screen "78_3BR" 800x454, template "Template_1"
   on GenerateScreen: SetTag("Tag_ScreenNumber", 78)
   TextField "Text field_1" at 17,28 size 250x21; Text 'Слово керування енкодером:'
   Circle "Circle_1" at 28,55 size 16x16
      Appearance <- "STW2_ENC"
   Circle "Circle_2" at 28,75 size 16x16
      Appearance <- "ZSW2_ENC"
   Circle "Circle_3" at 28,95 size 16x16
      Appearance <- "STW2_ENC"
   TextField "Text field_3" at 56,54 size 231x18; Text 'Трігер на калібровку енкодера'
   TextField "Text field_4" at 56,74 size 154x18; Text 'Квитування помилки'
   TextField "Text field_5" at 56,94 size 123x18; Text 'Контроль з PLC'
   IOField "I/O field_1" at 16,115 size 40x20; FormatPattern FFFF
      ProcessValue <- "STW2_ENC"
   TextField "Text field_6" at 56,115 size 248x18; Text 'Сигнал працездатності енкодера'
   TextField "Text field_12" at 403,28 size 210x21; Text 'Слово статусу енкодера:'
   Circle "Circle_9" at 414,55 size 16x16
      Appearance <- "ZSW2_ENC"
   TextField "Text field_14" at 442,54 size 350x18; Text 'Підтвердження встановлення нового значення'
   Circle "Circle_10" at 414,75 size 16x16
      Appearance <- "ZSW2_ENC"
   TextField "Text field_15" at 442,74 size 234x18; Text 'Фактичне положення є дійсним'
   Circle "Circle_11" at 414,95 size 16x16
      Appearance <- "ZSW2_ENC"
   TextField "Text field_16" at 442,94 size 228x18; Text 'Фактична швидкість є дійсною'
   Circle "Circle_12" at 414,115 size 16x16
      Appearance <- "ZSW2_ENC"
   TextField "Text field_17" at 442,114 size 129x18; Text 'Помилка активна'
   Circle "Circle_13" at 414,135 size 16x16
      Appearance <- "ZSW2_ENC"
   TextField "Text field_18" at 442,134 size 176x18; Text 'Попередження активне'
   Circle "Circle_14" at 414,155 size 16x16
      Appearance <- "ZSW2_ENC"
   TextField "Text field_19" at 442,154 size 145x18; Text 'Запит на перевірку'
   TextField "Text field_20" at 442,174 size 248x18; Text 'Сигнал працездатності енкодера'
   IOField "I/O field_2" at 402,173 size 40x20; FormatPattern FFFF
      ProcessValue <- "ZSW2_ENC"
   IOField "I/O field_3" at 148,364 size 70x20; FormatPattern s9999999999
      ProcessValue <- "RawPosition"
   TextField "Text field_26" at 28,363 size 107x21; Text 'Положення:'
   IOField "I/O field_4" at 534,364 size 70x20; FormatPattern s9999999999
      ProcessValue <- "RawVelocity"
   TextField "Text field_27" at 414,363 size 97x21; Text 'Швидкість:'
   Circle "Circle_4" at 28,222 size 16x16
      Appearance <- "EncoderLifeValid"
   TextField "Text field_2" at 56,221 size 228x18; Text 'Sign-of-life енкодера валідний'
   Circle "Circle_5" at 28,242 size 16x16
      Appearance <- "EncoderReady"
   TextField "Text field_7" at 56,241 size 325x18; Text 'Енкодер готовий для використання в логіці'
   Circle "Circle_6" at 28,262 size 16x16
      Appearance <- "CommunicationFault"
   TextField "Text field_8" at 56,261 size 288x18; Text 'Загальна помилка обміну з енкодером'
   Circle "Circle_7" at 28,282 size 16x16
      Appearance <- "PresetBusy"
   TextField "Text field_9" at 56,281 size 198x18; Text 'Preset-процедура активна'
   Circle "Circle_8" at 28,302 size 16x16
      Appearance <- "PresetDone"
   TextField "Text field_10" at 56,301 size 191x18; Text 'Preset успішно виконано.'
   Circle "Circle_15" at 28,322 size 16x16
      Appearance <- "PresetError"
   TextField "Text field_11" at 56,321 size 198x18; Text 'Помилка виконання preset'
   TextField "Text field_13" at 414,249 size 127x18; Text 'Статус енкодеру'
   TextField "Text field_21" at 414,221 size 115x18; Text 'Статус пресету'
   SymbolicIOField "Symbolic I/O field_1" at 562,214 size 230x32; TextOff '0'; TextOn '1'; TextList "PresetStatus"
      ProcessValue <- "PresetStatus"
   SymbolicIOField "Symbolic I/O field_2" at 562,242 size 230x32; TextOff '0'; TextOn '1'; TextList "EncoderStatus"
      ProcessValue <- "Status"
   TextField "Text field_22" at 308,6 size 185x23; Text 'Стан енкодеру 3BR'

screen "79_4BR1" 800x454, template "Template_1"
   on GenerateScreen: SetTag("Tag_ScreenNumber", 79)
   TextField "Text field_1" at 17,28 size 250x21; Text 'Слово керування енкодером:'
   Circle "Circle_1" at 28,55 size 16x16
      Appearance <- "STW2_ENC"
   Circle "Circle_2" at 28,75 size 16x16
      Appearance <- "ZSW2_ENC"
   Circle "Circle_3" at 28,95 size 16x16
      Appearance <- "STW2_ENC"
   TextField "Text field_3" at 56,54 size 231x18; Text 'Трігер на калібровку енкодера'
   TextField "Text field_4" at 56,74 size 154x18; Text 'Квитування помилки'
   TextField "Text field_5" at 56,94 size 123x18; Text 'Контроль з PLC'
   IOField "I/O field_1" at 16,115 size 40x20; FormatPattern FFFF
      ProcessValue <- "STW2_ENC"
   TextField "Text field_6" at 56,115 size 248x18; Text 'Сигнал працездатності енкодера'
   TextField "Text field_12" at 403,28 size 210x21; Text 'Слово статусу енкодера:'
   Circle "Circle_9" at 414,55 size 16x16
      Appearance <- "ZSW2_ENC"
   TextField "Text field_14" at 442,54 size 350x18; Text 'Підтвердження встановлення нового значення'
   Circle "Circle_10" at 414,75 size 16x16
      Appearance <- "ZSW2_ENC"
   TextField "Text field_15" at 442,74 size 234x18; Text 'Фактичне положення є дійсним'
   Circle "Circle_11" at 414,95 size 16x16
      Appearance <- "ZSW2_ENC"
   TextField "Text field_16" at 442,94 size 228x18; Text 'Фактична швидкість є дійсною'
   Circle "Circle_12" at 414,115 size 16x16
      Appearance <- "ZSW2_ENC"
   TextField "Text field_17" at 442,114 size 129x18; Text 'Помилка активна'
   Circle "Circle_13" at 414,135 size 16x16
      Appearance <- "ZSW2_ENC"
   TextField "Text field_18" at 442,134 size 176x18; Text 'Попередження активне'
   Circle "Circle_14" at 414,155 size 16x16
      Appearance <- "ZSW2_ENC"
   TextField "Text field_19" at 442,154 size 145x18; Text 'Запит на перевірку'
   TextField "Text field_20" at 442,174 size 248x18; Text 'Сигнал працездатності енкодера'
   IOField "I/O field_2" at 402,173 size 40x20; FormatPattern FFFF
      ProcessValue <- "ZSW2_ENC"
   IOField "I/O field_3" at 148,364 size 70x20; FormatPattern s9999999999
      ProcessValue <- "RawPosition"
   TextField "Text field_26" at 28,363 size 107x21; Text 'Положення:'
   IOField "I/O field_4" at 534,364 size 70x20; FormatPattern s9999999999
      ProcessValue <- "RawVelocity"
   TextField "Text field_27" at 414,363 size 97x21; Text 'Швидкість:'
   Circle "Circle_4" at 28,222 size 16x16
      Appearance <- "EncoderLifeValid"
   TextField "Text field_2" at 56,221 size 228x18; Text 'Sign-of-life енкодера валідний'
   Circle "Circle_5" at 28,242 size 16x16
      Appearance <- "EncoderReady"
   TextField "Text field_7" at 56,241 size 325x18; Text 'Енкодер готовий для використання в логіці'
   Circle "Circle_6" at 28,262 size 16x16
      Appearance <- "CommunicationFault"
   TextField "Text field_8" at 56,261 size 288x18; Text 'Загальна помилка обміну з енкодером'
   Circle "Circle_7" at 28,282 size 16x16
      Appearance <- "PresetBusy"
   TextField "Text field_9" at 56,281 size 198x18; Text 'Preset-процедура активна'
   Circle "Circle_8" at 28,302 size 16x16
      Appearance <- "PresetDone"
   TextField "Text field_10" at 56,301 size 191x18; Text 'Preset успішно виконано.'
   Circle "Circle_15" at 28,322 size 16x16
      Appearance <- "PresetError"
   TextField "Text field_11" at 56,321 size 198x18; Text 'Помилка виконання preset'
   TextField "Text field_13" at 414,249 size 127x18; Text 'Статус енкодеру'
   TextField "Text field_21" at 414,221 size 115x18; Text 'Статус пресету'
   SymbolicIOField "Symbolic I/O field_1" at 562,214 size 230x32; TextOff '0'; TextOn '1'; TextList "PresetStatus"
      ProcessValue <- "PresetStatus"
   SymbolicIOField "Symbolic I/O field_2" at 562,242 size 230x32; TextOff '0'; TextOn '1'; TextList "EncoderStatus"
      ProcessValue <- "Status"
   TextField "Text field_22" at 308,6 size 196x23; Text 'Стан енкодеру 4BR1'

screen "710_4BR2" 800x454, template "Template_1"
   on GenerateScreen: SetTag("Tag_ScreenNumber", 710)
   TextField "Text field_1" at 17,28 size 250x21; Text 'Слово керування енкодером:'
   Circle "Circle_1" at 28,55 size 16x16
      Appearance <- "STW2_ENC"
   Circle "Circle_2" at 28,75 size 16x16
      Appearance <- "ZSW2_ENC"
   Circle "Circle_3" at 28,95 size 16x16
      Appearance <- "STW2_ENC"
   TextField "Text field_3" at 56,54 size 231x18; Text 'Трігер на калібровку енкодера'
   TextField "Text field_4" at 56,74 size 154x18; Text 'Квитування помилки'
   TextField "Text field_5" at 56,94 size 123x18; Text 'Контроль з PLC'
   IOField "I/O field_1" at 16,115 size 40x20; FormatPattern FFFF
      ProcessValue <- "STW2_ENC"
   TextField "Text field_6" at 56,115 size 248x18; Text 'Сигнал працездатності енкодера'
   TextField "Text field_12" at 403,28 size 210x21; Text 'Слово статусу енкодера:'
   Circle "Circle_9" at 414,55 size 16x16
      Appearance <- "ZSW2_ENC"
   TextField "Text field_14" at 442,54 size 350x18; Text 'Підтвердження встановлення нового значення'
   Circle "Circle_10" at 414,75 size 16x16
      Appearance <- "ZSW2_ENC"
   TextField "Text field_15" at 442,74 size 234x18; Text 'Фактичне положення є дійсним'
   Circle "Circle_11" at 414,95 size 16x16
      Appearance <- "ZSW2_ENC"
   TextField "Text field_16" at 442,94 size 228x18; Text 'Фактична швидкість є дійсною'
   Circle "Circle_12" at 414,115 size 16x16
      Appearance <- "ZSW2_ENC"
   TextField "Text field_17" at 442,114 size 129x18; Text 'Помилка активна'
   Circle "Circle_13" at 414,135 size 16x16
      Appearance <- "ZSW2_ENC"
   TextField "Text field_18" at 442,134 size 176x18; Text 'Попередження активне'
   Circle "Circle_14" at 414,155 size 16x16
      Appearance <- "ZSW2_ENC"
   TextField "Text field_19" at 442,154 size 145x18; Text 'Запит на перевірку'
   TextField "Text field_20" at 442,174 size 248x18; Text 'Сигнал працездатності енкодера'
   IOField "I/O field_2" at 402,173 size 40x20; FormatPattern FFFF
      ProcessValue <- "ZSW2_ENC"
   IOField "I/O field_3" at 148,364 size 70x20; FormatPattern s9999999999
      ProcessValue <- "RawPosition"
   TextField "Text field_26" at 28,363 size 107x21; Text 'Положення:'
   IOField "I/O field_4" at 534,364 size 70x20; FormatPattern s9999999999
      ProcessValue <- "RawVelocity"
   TextField "Text field_27" at 414,363 size 97x21; Text 'Швидкість:'
   Circle "Circle_4" at 28,222 size 16x16
      Appearance <- "EncoderLifeValid"
   TextField "Text field_2" at 56,221 size 228x18; Text 'Sign-of-life енкодера валідний'
   Circle "Circle_5" at 28,242 size 16x16
      Appearance <- "EncoderReady"
   TextField "Text field_7" at 56,241 size 325x18; Text 'Енкодер готовий для використання в логіці'
   Circle "Circle_6" at 28,262 size 16x16
      Appearance <- "CommunicationFault"
   TextField "Text field_8" at 56,261 size 288x18; Text 'Загальна помилка обміну з енкодером'
   Circle "Circle_7" at 28,282 size 16x16
      Appearance <- "PresetBusy"
   TextField "Text field_9" at 56,281 size 198x18; Text 'Preset-процедура активна'
   Circle "Circle_8" at 28,302 size 16x16
      Appearance <- "PresetDone"
   TextField "Text field_10" at 56,301 size 191x18; Text 'Preset успішно виконано.'
   Circle "Circle_15" at 28,322 size 16x16
      Appearance <- "PresetError"
   TextField "Text field_11" at 56,321 size 198x18; Text 'Помилка виконання preset'
   TextField "Text field_13" at 414,249 size 127x18; Text 'Статус енкодеру'
   TextField "Text field_21" at 414,221 size 115x18; Text 'Статус пресету'
   SymbolicIOField "Symbolic I/O field_1" at 562,214 size 230x32; TextOff '0'; TextOn '1'; TextList "PresetStatus"
      ProcessValue <- "PresetStatus"
   SymbolicIOField "Symbolic I/O field_2" at 562,242 size 230x32; TextOff '0'; TextOn '1'; TextList "EncoderStatus"
      ProcessValue <- "Status"
   TextField "Text field_22" at 308,6 size 196x23; Text 'Стан енкодеру 4BR2'

screen "61_Архіви(3UZ1)" 800x454, template "Template_1"
   on GenerateScreen: SetTag("Tag_ScreenNumber", 61); SetTag("iVisibilityDevices", 0)
   Button "btnLiftUp" at 8,120 size 96x32; TextOff '3UZ1'
   Button "btnTrolley" at 8,160 size 96x32; TextOff '4UZ1'
      on Release: ActivateScreen("62_Архіви(4UZ1)", 0)
   Button "btnCrane" at 8,200 size 96x32; TextOff '4UZ2'
      on Release: ActivateScreen("63_Архіви(4UZ2)", 0)
   Button "btnContactor" at 8,80 size 96x32; TextOff '1UZ1'
      on Release: ActivateScreen("60_Архіви(1UZ1)", 0)
   Button "Button_1" at 8,319 size 96x32; TextOff 'Струм Момент'
      on Release: SetTag("iVisibilityDevices", 0)
      Appearance <- "iVisibilityDevices"
   Button "Button_2" at 8,356 size 96x32; TextOff 'Швидкості'
      on Release: SetTag("iVisibilityDevices", 1)
      Appearance <- "iVisibilityDevices"
   TrendView "trvCurrent" at 155,10 size 640x200
      Visibility <- "iVisibilityDevices"
   TrendView "trvMoment" at 155,208 size 640x200
      Visibility <- "iVisibilityDevices"
   TextField "txtCurrent" at 125,95 size 19x30; Text 'I ,А'
      Visibility <- "iVisibilityDevices"
   TextField "txtMoment" at 125,278 size 19x60; Text 'M , Н*м'
      Visibility <- "iVisibilityDevices"
   Button "btnCurrentDoubleBack" at 111,10 size 40x20; TextOff 'Text'; PictureOff "FB_2ArrowsLeft_Rectangular_Released_256c"; PictureOn "FB_2ArrowsLeft_Rectangular_Pressed_256c"
      on Press: function_f26ff0ec("trvCurrent")
      on Release: function_f26ff0ec("trvCurrent")
      Visibility <- "iVisibilityDevices"
   Button "btnCurrentOneBack" at 111,35 size 40x20; TextOff 'Text'; PictureOff "FB_ArrowLeft_Rectangular_Released_256c"; PictureOn "FB_ArrowLeft_Rectangular_Pressed_256c"
      on Press: function_f26ff0ec("trvCurrent")
      Visibility <- "iVisibilityDevices"
   Button "btnCurrentForward" at 111,149 size 40x20; TextOff 'Text'; PictureOff "FB_ArrowRight_Rectangular_Released_256c"; PictureOn "FB_ArrowRight_Rectangular_Pressed_256c"
      on Press: function_c2ce674d("trvCurrent")
      Visibility <- "iVisibilityDevices"
   Button "btnCurrentDoubleForward" at 111,174 size 40x20; TextOff 'Text'; PictureOff "FB_2ArrowsRight_Rectangular_Released_256c"; PictureOn "FB_2ArrowsRight_Rectangular_Pressed_256c"
      on Press: function_c2ce674d("trvCurrent")
      on Release: function_c2ce674d("trvCurrent")
      Visibility <- "iVisibilityDevices"
   Button "btnMomentDoubleBack" at 111,208 size 40x20; TextOff 'Text'; PictureOff "FB_2ArrowsLeft_Rectangular_Released_256c"; PictureOn "FB_2ArrowsLeft_Rectangular_Pressed_256c"
      on Press: function_f26ff0ec("trvMoment")
      on Release: function_f26ff0ec("trvMoment")
      Visibility <- "iVisibilityDevices"
   Button "btnMomentOneBack" at 111,233 size 40x20; TextOff 'Text'; PictureOff "FB_ArrowLeft_Rectangular_Released_256c"; PictureOn "FB_ArrowLeft_Rectangular_Pressed_256c"
      on Press: function_f26ff0ec("trvMoment")
      Visibility <- "iVisibilityDevices"
   Button "btnMomentOneForward" at 111,363 size 40x20; TextOff 'Text'; PictureOff "FB_ArrowRight_Rectangular_Released_256c"; PictureOn "FB_ArrowRight_Rectangular_Pressed_256c"
      on Press: function_c2ce674d("trvMoment")
      Visibility <- "iVisibilityDevices"
   Button "btnMomentDoubleForward" at 111,388 size 40x20; TextOff 'Text'; PictureOff "FB_2ArrowsRight_Rectangular_Released_256c"; PictureOn "FB_2ArrowsRight_Rectangular_Pressed_256c"
      on Press: function_c2ce674d("trvMoment")
      on Release: function_c2ce674d("trvMoment")
      Visibility <- "iVisibilityDevices"
   TrendView "trvSpeed" at 155,10 size 640x200
      Visibility <- "iVisibilityDevices"
   TrendView "trvError" at 155,208 size 640x200
      Visibility <- "iVisibilityDevices"
   TextField "txtSpeed" at 108,84 size 19x53; Text 'W_set,'
      Visibility <- "iVisibilityDevices"
   TextField "txtError" at 125,259 size 19x98; Text 'W_err ,об/хв'
      Visibility <- "iVisibilityDevices"
   TextField "txtSpeed_1" at 120,82 size 19x57; Text 'W_real,'
      Visibility <- "iVisibilityDevices"
   TextField "txtSpeed_2" at 132,87 size 19x46; Text 'об/хв'
      Visibility <- "iVisibilityDevices"
   Button "btnSpeedDoubleBack" at 111,10 size 40x20; TextOff 'Text'; PictureOff "FB_2ArrowsLeft_Rectangular_Released_256c"; PictureOn "FB_2ArrowsLeft_Rectangular_Pressed_256c"
      on Press: function_f26ff0ec("trvSpeed")
      on Release: function_f26ff0ec("trvSpeed")
      Visibility <- "iVisibilityDevices"
   Button "btnSpeedOneBack" at 111,35 size 40x20; TextOff 'Text'; PictureOff "FB_ArrowLeft_Rectangular_Released_256c"; PictureOn "FB_ArrowLeft_Rectangular_Pressed_256c"
      on Press: function_f26ff0ec("trvSpeed")
      Visibility <- "iVisibilityDevices"
   Button "btnSpeedForward" at 111,149 size 40x20; TextOff 'Text'; PictureOff "FB_ArrowRight_Rectangular_Released_256c"; PictureOn "FB_ArrowRight_Rectangular_Pressed_256c"
      on Press: function_c2ce674d("trvSpeed")
      Visibility <- "iVisibilityDevices"
   Button "btnSpeedDoubleForward" at 111,174 size 40x20; TextOff 'Text'; PictureOff "FB_2ArrowsRight_Rectangular_Released_256c"; PictureOn "FB_2ArrowsRight_Rectangular_Pressed_256c"
      on Press: function_c2ce674d("trvSpeed")
      on Release: function_c2ce674d("trvSpeed")
      Visibility <- "iVisibilityDevices"
   Button "btnErrorDoubleBack" at 111,208 size 40x20; TextOff 'Text'; PictureOff "FB_2ArrowsLeft_Rectangular_Released_256c"; PictureOn "FB_2ArrowsLeft_Rectangular_Pressed_256c"
      on Press: function_f26ff0ec("trvError")
      on Release: function_f26ff0ec("trvError")
      Visibility <- "iVisibilityDevices"
   Button "btnErrorOneBack" at 111,233 size 40x20; TextOff 'Text'; PictureOff "FB_ArrowLeft_Rectangular_Released_256c"; PictureOn "FB_ArrowLeft_Rectangular_Pressed_256c"
      on Press: function_f26ff0ec("trvError")
      Visibility <- "iVisibilityDevices"
   Button "btnErrorOneForward" at 111,363 size 40x20; TextOff 'Text'; PictureOff "FB_ArrowRight_Rectangular_Released_256c"; PictureOn "FB_ArrowRight_Rectangular_Pressed_256c"
      on Press: function_c2ce674d("trvError")
      Visibility <- "iVisibilityDevices"
   Button "btnErrorDoubleForward" at 111,388 size 40x20; TextOff 'Text'; PictureOff "FB_2ArrowsRight_Rectangular_Released_256c"; PictureOn "FB_2ArrowsRight_Rectangular_Pressed_256c"
      on Press: function_c2ce674d("trvError")
      on Release: function_c2ce674d("trvError")
      Visibility <- "iVisibilityDevices"

screen "62_Архіви(4UZ1)" 800x454, template "Template_1"
   on GenerateScreen: SetTag("Tag_ScreenNumber", 62); SetTag("iVisibilityDevices", 0)
   Button "btnLiftUp" at 8,120 size 96x32; TextOff '3UZ1'
      on Release: ActivateScreen("61_Архіви(3UZ1)", 0)
   Button "btnTrolley" at 8,160 size 96x32; TextOff '4UZ1'
   Button "btnCrane" at 8,200 size 96x32; TextOff '4UZ2'
      on Release: ActivateScreen("63_Архіви(4UZ2)", 0)
   Button "btnContactor" at 8,80 size 96x32; TextOff '1UZ1'
      on Release: ActivateScreen("60_Архіви(1UZ1)", 0)
   Button "Button_1" at 8,319 size 96x32; TextOff 'Струм Момент'
      on Release: SetTag("iVisibilityDevices", 0)
      Appearance <- "iVisibilityDevices"
   Button "Button_2" at 8,356 size 96x32; TextOff 'Швидкості'
      on Release: SetTag("iVisibilityDevices", 1)
      Appearance <- "iVisibilityDevices"
   TrendView "trvCurrent" at 155,10 size 640x200
      Visibility <- "iVisibilityDevices"
   TrendView "trvMoment" at 155,208 size 640x200
      Visibility <- "iVisibilityDevices"
   TextField "txtCurrent" at 125,95 size 19x30; Text 'I ,А'
      Visibility <- "iVisibilityDevices"
   TextField "txtMoment" at 125,278 size 19x60; Text 'M , Н*м'
      Visibility <- "iVisibilityDevices"
   Button "btnCurrentDoubleBack" at 111,10 size 40x20; TextOff 'Text'; PictureOff "FB_2ArrowsLeft_Rectangular_Released_256c"; PictureOn "FB_2ArrowsLeft_Rectangular_Pressed_256c"
      on Press: function_f26ff0ec("trvCurrent")
      on Release: function_f26ff0ec("trvCurrent")
      Visibility <- "iVisibilityDevices"
   Button "btnCurrentOneBack" at 111,35 size 40x20; TextOff 'Text'; PictureOff "FB_ArrowLeft_Rectangular_Released_256c"; PictureOn "FB_ArrowLeft_Rectangular_Pressed_256c"
      on Press: function_f26ff0ec("trvCurrent")
      Visibility <- "iVisibilityDevices"
   Button "btnCurrentForward" at 111,149 size 40x20; TextOff 'Text'; PictureOff "FB_ArrowRight_Rectangular_Released_256c"; PictureOn "FB_ArrowRight_Rectangular_Pressed_256c"
      on Press: function_c2ce674d("trvCurrent")
      Visibility <- "iVisibilityDevices"
   Button "btnCurrentDoubleForward" at 111,174 size 40x20; TextOff 'Text'; PictureOff "FB_2ArrowsRight_Rectangular_Released_256c"; PictureOn "FB_2ArrowsRight_Rectangular_Pressed_256c"
      on Press: function_c2ce674d("trvCurrent")
      on Release: function_c2ce674d("trvCurrent")
      Visibility <- "iVisibilityDevices"
   Button "btnMomentDoubleBack" at 111,208 size 40x20; TextOff 'Text'; PictureOff "FB_2ArrowsLeft_Rectangular_Released_256c"; PictureOn "FB_2ArrowsLeft_Rectangular_Pressed_256c"
      on Press: function_f26ff0ec("trvMoment")
      on Release: function_f26ff0ec("trvMoment")
      Visibility <- "iVisibilityDevices"
   Button "btnMomentOneBack" at 111,233 size 40x20; TextOff 'Text'; PictureOff "FB_ArrowLeft_Rectangular_Released_256c"; PictureOn "FB_ArrowLeft_Rectangular_Pressed_256c"
      on Press: function_f26ff0ec("trvMoment")
      Visibility <- "iVisibilityDevices"
   Button "btnMomentOneForward" at 111,363 size 40x20; TextOff 'Text'; PictureOff "FB_ArrowRight_Rectangular_Released_256c"; PictureOn "FB_ArrowRight_Rectangular_Pressed_256c"
      on Press: function_c2ce674d("trvMoment")
      Visibility <- "iVisibilityDevices"
   Button "btnMomentDoubleForward" at 111,388 size 40x20; TextOff 'Text'; PictureOff "FB_2ArrowsRight_Rectangular_Released_256c"; PictureOn "FB_2ArrowsRight_Rectangular_Pressed_256c"
      on Press: function_c2ce674d("trvMoment")
      on Release: function_c2ce674d("trvMoment")
      Visibility <- "iVisibilityDevices"
   TrendView "trvSpeed" at 155,10 size 640x200
      Visibility <- "iVisibilityDevices"
   TrendView "trvError" at 155,208 size 640x200
      Visibility <- "iVisibilityDevices"
   TextField "txtSpeed" at 108,84 size 19x53; Text 'W_set,'
      Visibility <- "iVisibilityDevices"
   TextField "txtError" at 125,259 size 19x98; Text 'W_err ,об/хв'
      Visibility <- "iVisibilityDevices"
   TextField "txtSpeed_1" at 120,82 size 19x57; Text 'W_real,'
      Visibility <- "iVisibilityDevices"
   TextField "txtSpeed_2" at 132,87 size 19x46; Text 'об/хв'
      Visibility <- "iVisibilityDevices"
   Button "btnSpeedDoubleBack" at 111,10 size 40x20; TextOff 'Text'; PictureOff "FB_2ArrowsLeft_Rectangular_Released_256c"; PictureOn "FB_2ArrowsLeft_Rectangular_Pressed_256c"
      on Press: function_f26ff0ec("trvSpeed")
      on Release: function_f26ff0ec("trvSpeed")
      Visibility <- "iVisibilityDevices"
   Button "btnSpeedOneBack" at 111,35 size 40x20; TextOff 'Text'; PictureOff "FB_ArrowLeft_Rectangular_Released_256c"; PictureOn "FB_ArrowLeft_Rectangular_Pressed_256c"
      on Press: function_f26ff0ec("trvSpeed")
      Visibility <- "iVisibilityDevices"
   Button "btnSpeedForward" at 111,149 size 40x20; TextOff 'Text'; PictureOff "FB_ArrowRight_Rectangular_Released_256c"; PictureOn "FB_ArrowRight_Rectangular_Pressed_256c"
      on Press: function_c2ce674d("trvSpeed")
      Visibility <- "iVisibilityDevices"
   Button "btnSpeedDoubleForward" at 111,174 size 40x20; TextOff 'Text'; PictureOff "FB_2ArrowsRight_Rectangular_Released_256c"; PictureOn "FB_2ArrowsRight_Rectangular_Pressed_256c"
      on Press: function_c2ce674d("trvSpeed")
      on Release: function_c2ce674d("trvSpeed")
      Visibility <- "iVisibilityDevices"
   Button "btnErrorDoubleBack" at 111,208 size 40x20; TextOff 'Text'; PictureOff "FB_2ArrowsLeft_Rectangular_Released_256c"; PictureOn "FB_2ArrowsLeft_Rectangular_Pressed_256c"
      on Press: function_f26ff0ec("trvError")
      on Release: function_f26ff0ec("trvError")
      Visibility <- "iVisibilityDevices"
   Button "btnErrorOneBack" at 111,233 size 40x20; TextOff 'Text'; PictureOff "FB_ArrowLeft_Rectangular_Released_256c"; PictureOn "FB_ArrowLeft_Rectangular_Pressed_256c"
      on Press: function_f26ff0ec("trvError")
      Visibility <- "iVisibilityDevices"
   Button "btnErrorOneForward" at 111,363 size 40x20; TextOff 'Text'; PictureOff "FB_ArrowRight_Rectangular_Released_256c"; PictureOn "FB_ArrowRight_Rectangular_Pressed_256c"
      on Press: function_c2ce674d("trvError")
      Visibility <- "iVisibilityDevices"
   Button "btnErrorDoubleForward" at 111,388 size 40x20; TextOff 'Text'; PictureOff "FB_2ArrowsRight_Rectangular_Released_256c"; PictureOn "FB_2ArrowsRight_Rectangular_Pressed_256c"
      on Press: function_c2ce674d("trvError")
      on Release: function_c2ce674d("trvError")
      Visibility <- "iVisibilityDevices"

screen "63_Архіви(4UZ2)" 800x454, template "Template_1"
   on GenerateScreen: SetTag("Tag_ScreenNumber", 63); SetTag("iVisibilityDevices", 0)
   Button "btnLiftUp" at 8,120 size 96x32; TextOff '3UZ1'
      on Release: ActivateScreen("61_Архіви(3UZ1)", 0)
   Button "btnTrolley" at 8,160 size 96x32; TextOff '4UZ1'
      on Release: ActivateScreen("62_Архіви(4UZ1)", 0)
   Button "btnCrane" at 8,200 size 96x32; TextOff '4UZ2'
   Button "btnContactor" at 8,80 size 96x32; TextOff '1UZ1'
      on Release: ActivateScreen("60_Архіви(1UZ1)", 0)
   Button "Button_1" at 8,319 size 96x32; TextOff 'Струм Момент'
      on Release: SetTag("iVisibilityDevices", 0)
      Appearance <- "iVisibilityDevices"
   Button "Button_2" at 8,356 size 96x32; TextOff 'Швидкості'
      on Release: SetTag("iVisibilityDevices", 1)
      Appearance <- "iVisibilityDevices"
   TrendView "trvCurrent" at 155,10 size 640x200
      Visibility <- "iVisibilityDevices"
   TrendView "trvMoment" at 155,208 size 640x200
      Visibility <- "iVisibilityDevices"
   TextField "txtCurrent" at 125,95 size 19x30; Text 'I ,А'
      Visibility <- "iVisibilityDevices"
   TextField "txtMoment" at 125,278 size 19x60; Text 'M , Н*м'
      Visibility <- "iVisibilityDevices"
   Button "btnCurrentDoubleBack" at 111,10 size 40x20; TextOff 'Text'; PictureOff "FB_2ArrowsLeft_Rectangular_Released_256c"; PictureOn "FB_2ArrowsLeft_Rectangular_Pressed_256c"
      on Press: function_f26ff0ec("trvCurrent")
      on Release: function_f26ff0ec("trvCurrent")
      Visibility <- "iVisibilityDevices"
   Button "btnCurrentOneBack" at 111,35 size 40x20; TextOff 'Text'; PictureOff "FB_ArrowLeft_Rectangular_Released_256c"; PictureOn "FB_ArrowLeft_Rectangular_Pressed_256c"
      on Press: function_f26ff0ec("trvCurrent")
      Visibility <- "iVisibilityDevices"
   Button "btnCurrentForward" at 111,149 size 40x20; TextOff 'Text'; PictureOff "FB_ArrowRight_Rectangular_Released_256c"; PictureOn "FB_ArrowRight_Rectangular_Pressed_256c"
      on Press: function_c2ce674d("trvCurrent")
      Visibility <- "iVisibilityDevices"
   Button "btnCurrentDoubleForward" at 111,174 size 40x20; TextOff 'Text'; PictureOff "FB_2ArrowsRight_Rectangular_Released_256c"; PictureOn "FB_2ArrowsRight_Rectangular_Pressed_256c"
      on Press: function_c2ce674d("trvCurrent")
      on Release: function_c2ce674d("trvCurrent")
      Visibility <- "iVisibilityDevices"
   Button "btnMomentDoubleBack" at 111,208 size 40x20; TextOff 'Text'; PictureOff "FB_2ArrowsLeft_Rectangular_Released_256c"; PictureOn "FB_2ArrowsLeft_Rectangular_Pressed_256c"
      on Press: function_f26ff0ec("trvMoment")
      on Release: function_f26ff0ec("trvMoment")
      Visibility <- "iVisibilityDevices"
   Button "btnMomentOneBack" at 111,233 size 40x20; TextOff 'Text'; PictureOff "FB_ArrowLeft_Rectangular_Released_256c"; PictureOn "FB_ArrowLeft_Rectangular_Pressed_256c"
      on Press: function_f26ff0ec("trvMoment")
      Visibility <- "iVisibilityDevices"
   Button "btnMomentOneForward" at 111,363 size 40x20; TextOff 'Text'; PictureOff "FB_ArrowRight_Rectangular_Released_256c"; PictureOn "FB_ArrowRight_Rectangular_Pressed_256c"
      on Press: function_c2ce674d("trvMoment")
      Visibility <- "iVisibilityDevices"
   Button "btnMomentDoubleForward" at 111,388 size 40x20; TextOff 'Text'; PictureOff "FB_2ArrowsRight_Rectangular_Released_256c"; PictureOn "FB_2ArrowsRight_Rectangular_Pressed_256c"
      on Press: function_c2ce674d("trvMoment")
      on Release: function_c2ce674d("trvMoment")
      Visibility <- "iVisibilityDevices"
   TrendView "trvSpeed" at 155,10 size 640x200
      Visibility <- "iVisibilityDevices"
   TrendView "trvError" at 155,208 size 640x200
      Visibility <- "iVisibilityDevices"
   TextField "txtSpeed" at 108,84 size 19x53; Text 'W_set,'
      Visibility <- "iVisibilityDevices"
   TextField "txtError" at 125,259 size 19x98; Text 'W_err ,об/хв'
      Visibility <- "iVisibilityDevices"
   TextField "txtSpeed_1" at 120,82 size 19x57; Text 'W_real,'
      Visibility <- "iVisibilityDevices"
   TextField "txtSpeed_2" at 132,87 size 19x46; Text 'об/хв'
      Visibility <- "iVisibilityDevices"
   Button "btnSpeedDoubleBack" at 111,10 size 40x20; TextOff 'Text'; PictureOff "FB_2ArrowsLeft_Rectangular_Released_256c"; PictureOn "FB_2ArrowsLeft_Rectangular_Pressed_256c"
      on Press: function_f26ff0ec("trvSpeed")
      on Release: function_f26ff0ec("trvSpeed")
      Visibility <- "iVisibilityDevices"
   Button "btnSpeedOneBack" at 111,35 size 40x20; TextOff 'Text'; PictureOff "FB_ArrowLeft_Rectangular_Released_256c"; PictureOn "FB_ArrowLeft_Rectangular_Pressed_256c"
      on Press: function_f26ff0ec("trvSpeed")
      Visibility <- "iVisibilityDevices"
   Button "btnSpeedForward" at 111,149 size 40x20; TextOff 'Text'; PictureOff "FB_ArrowRight_Rectangular_Released_256c"; PictureOn "FB_ArrowRight_Rectangular_Pressed_256c"
      on Press: function_c2ce674d("trvSpeed")
      Visibility <- "iVisibilityDevices"
   Button "btnSpeedDoubleForward" at 111,174 size 40x20; TextOff 'Text'; PictureOff "FB_2ArrowsRight_Rectangular_Released_256c"; PictureOn "FB_2ArrowsRight_Rectangular_Pressed_256c"
      on Press: function_c2ce674d("trvSpeed")
      on Release: function_c2ce674d("trvSpeed")
      Visibility <- "iVisibilityDevices"
   Button "btnErrorDoubleBack" at 111,208 size 40x20; TextOff 'Text'; PictureOff "FB_2ArrowsLeft_Rectangular_Released_256c"; PictureOn "FB_2ArrowsLeft_Rectangular_Pressed_256c"
      on Press: function_f26ff0ec("trvError")
      on Release: function_f26ff0ec("trvError")
      Visibility <- "iVisibilityDevices"
   Button "btnErrorOneBack" at 111,233 size 40x20; TextOff 'Text'; PictureOff "FB_ArrowLeft_Rectangular_Released_256c"; PictureOn "FB_ArrowLeft_Rectangular_Pressed_256c"
      on Press: function_f26ff0ec("trvError")
      Visibility <- "iVisibilityDevices"
   Button "btnErrorOneForward" at 111,363 size 40x20; TextOff 'Text'; PictureOff "FB_ArrowRight_Rectangular_Released_256c"; PictureOn "FB_ArrowRight_Rectangular_Pressed_256c"
      on Press: function_c2ce674d("trvError")
      Visibility <- "iVisibilityDevices"
   Button "btnErrorDoubleForward" at 111,388 size 40x20; TextOff 'Text'; PictureOff "FB_2ArrowsRight_Rectangular_Released_256c"; PictureOn "FB_2ArrowsRight_Rectangular_Pressed_256c"
      on Press: function_c2ce674d("trvError")
      on Release: function_c2ce674d("trvError")
      Visibility <- "iVisibilityDevices"

screen "80_Калібровка" 800x454, template "Template_1"
   on GenerateScreen: SetTag("Tag_ScreenNumber", 80)
   Button "Button_1" at 305,160 size 85x25; TextOff 'Детальніше'
      on Release: ActivateScreen("81_КалібровкаПідйому", 0)
   Button "Button_2" at 705,160 size 85x25; TextOff 'Детальніше'
      on Release: ActivateScreen("82_КалібровкаВізка", 0)
   Button "Button_3" at 704,374 size 85x25; TextOff 'Детальніше'
      on Release: ActivateScreen("83_КалібровкаКрану", 0)
   TextField "Text field_1" at 20,13 size 157x21; Text 'Механізм підйому:'
   Circle "Circle_40" at 30,40 size 16x16
      Appearance <- "HMI_DB_Calibration_Hoist_Diagnostics_EncoderControlHealthy"
   TextField "Text field_40" at 58,39 size 335x18; Text 'Справність контролю 1BR'
   Circle "Circle_21" at 30,60 size 16x16
      Appearance <- "HMI_DB_Calibration_Hoist_Diagnostics_StartupDataConsistent"
   TextField "Text field_21" at 58,59 size 335x18; Text 'Контроль узгодженості даних після увімк. ПЛК'
   Circle "Circle_22" at 30,80 size 16x16
      Appearance <- "HMI_DB_Calibration_Hoist_Diagnostics_NoMovementWithoutCommand"
   TextField "Text field_22" at 58,79 size 335x18; Text 'Контроль коректності значень без команди руху'
   Circle "Circle_1" at 30,100 size 16x16
      Appearance <- "HMI_DB_Calibration_Hoist_Diagnostics_NoManualMovementDetected"
   TextField "Text field_2" at 58,99 size 335x18; Text 'Контроль коректності без активації ручн. приводу'
   Circle "Circle_2" at 30,120 size 16x16
      Appearance <- "HMI_DB_Calibration_Hoist_Diagnostics_EncoderUpdatesDuringMotion"
   TextField "Text field_6" at 58,119 size 290x18; Text 'Контроль оновлення значень під час руху'
   Circle "Circle_3" at 30,140 size 16x16
      Appearance <- "HMI_DB_Calibration_Hoist_Diagnostics_EncoderReplacementNotDetected"
   TextField "Text field_3" at 58,139 size 250x18; Text 'Контроль фізичної заміни енкодера'
   TextField "Text field_4" at 420,13 size 130x21; Text 'Механізм візка:'
   Circle "Circle_4" at 430,40 size 16x16
      Appearance <- "HMI_DB_Calibration_Trolley_Diagnostics_EncoderControlHealthy"
   TextField "Text field_5" at 458,39 size 335x18; Text 'Справність контролю 3BR'
   Circle "Circle_5" at 430,60 size 16x16
      Appearance <- "HMI_DB_Calibration_Trolley_Diagnostics_StartupDataConsistent"
   TextField "Text field_7" at 458,59 size 335x18; Text 'Контроль узгодженості даних після увімк. ПЛК'
   Circle "Circle_6" at 430,80 size 16x16
      Appearance <- "HMI_DB_Calibration_Trolley_Diagnostics_NoMovementWithoutCommand"
   TextField "Text field_8" at 458,79 size 335x18; Text 'Контроль коректності значень без команди руху'
   Circle "Circle_7" at 430,100 size 16x16
      Appearance <- "HMI_DB_Calibration_Trolley_Diagnostics_NoManualMovementDetected"
   TextField "Text field_9" at 458,99 size 335x18; Text 'Контроль коректності без активації ручн. приводу'
   Circle "Circle_8" at 430,120 size 16x16
      Appearance <- "HMI_DB_Calibration_Trolley_Diagnostics_EncoderUpdatesDuringMotion"
   TextField "Text field_10" at 458,119 size 335x18; Text 'Контроль оновлення значень під час руху'
   Circle "Circle_9" at 430,140 size 16x16
      Appearance <- "HMI_DB_Calibration_Trolley_Diagnostics_EncoderReplacementNotDetected"
   TextField "Text field_11" at 458,139 size 250x18; Text 'Контроль фізичної заміни енкодера'
   TextField "Text field_12" at 20,200 size 157x21; Text 'Механізм моста: / Механізм підйому:'
   Circle "Circle_10" at 30,227 size 16x16
      Appearance <- "HMI_DB_Calibration_Crane_Diagnostics_Encoder1ControlHealthy"
   TextField "Text field_13" at 58,226 size 335x18; Text 'Справність контролю 4BR1'
   Circle "Circle_11" at 30,247 size 16x16
      Appearance <- "HMI_DB_Calibration_Crane_Diagnostics_Encoder1StartupDataConsistent"
   TextField "Text field_14" at 58,246 size 335x18; Text 'Контроль узгодженості даних після увімк. ПЛК'
   Circle "Circle_12" at 30,267 size 16x16
      Appearance <- "HMI_DB_Calibration_Crane_Diagnostics_Encoder1NoMovementWithoutCommand"
   TextField "Text field_15" at 58,266 size 335x18; Text 'Контроль коректності значень без команди руху'
   Circle "Circle_13" at 30,287 size 16x16
      Appearance <- "HMI_DB_Calibration_Crane_Diagnostics_Encoder1NoManualMovementDetected"
   TextField "Text field_16" at 58,286 size 335x18; Text 'Контроль коректності без активації ручн. приводу'
   Circle "Circle_14" at 30,307 size 16x16
      Appearance <- "HMI_DB_Calibration_Crane_Diagnostics_Encoder1UpdatesDuringMotion"
   TextField "Text field_17" at 58,306 size 335x18; Text 'Контроль оновлення значень під час руху'
   Circle "Circle_15" at 30,327 size 16x16
      Appearance <- "HMI_DB_Calibration_Crane_Diagnostics_Encoder1ReplacementNotDetected"
   TextField "Text field_18" at 58,326 size 335x18; Text 'Контроль фізичної заміни енкодера'
   Circle "Circle_16" at 430,227 size 16x16
      Appearance <- "HMI_DB_Calibration_Crane_Diagnostics_Encoder2ControlHealthy"
   TextField "Text field_19" at 458,226 size 335x18; Text 'Справність контролю 4BR2'
   Circle "Circle_17" at 430,247 size 16x16
      Appearance <- "HMI_DB_Calibration_Crane_Diagnostics_Encoder2StartupDataConsistent"
   TextField "Text field_20" at 458,246 size 335x18; Text 'Контроль узгодженості даних після увімк. ПЛК'
   Circle "Circle_18" at 430,267 size 16x16
      Appearance <- "HMI_DB_Calibration_Crane_Diagnostics_Encoder2NoMovementWithoutCommand"
   TextField "Text field_23" at 458,266 size 335x18; Text 'Контроль коректності значень без команди руху'
   Circle "Circle_19" at 430,287 size 16x16
      Appearance <- "HMI_DB_Calibration_Crane_Diagnostics_Encoder2NoManualMovementDetected"
   TextField "Text field_24" at 458,286 size 335x18; Text 'Контроль коректності без активації ручн. приводу'
   Circle "Circle_20" at 430,307 size 16x16
      Appearance <- "HMI_DB_Calibration_Crane_Diagnostics_Encoder2UpdatesDuringMotion"
   TextField "Text field_25" at 458,306 size 335x18; Text 'Контроль оновлення значень під час руху'
   Circle "Circle_23" at 430,327 size 16x16
      Appearance <- "HMI_DB_Calibration_Crane_Diagnostics_Encoder2ReplacementNotDetected"
   TextField "Text field_26" at 458,326 size 335x18; Text 'Контроль фізичної заміни енкодера'
   Circle "Circle_24" at 262,380 size 16x16
      Appearance <- "HMI_DB_Calibration_Crane_Calibrated"
   TextField "Text field_27" at 290,379 size 335x18; Text 'Калібровка механізму / Розбіжності даних на енкодерах моста'
   Circle "Circle_25" at 30,160 size 16x16
      Appearance <- "HMI_DB_Calibration_Hoist_Calibrated"
   TextField "Text field_28" at 58,159 size 200x18; Text 'Контроль фізичної заміни енкодера / Калібровка механізму'
   Circle "Circle_26" at 430,160 size 16x16
      Appearance <- "HMI_DB_Calibration_Trolley_Calibrated"
   TextField "Text field_29" at 458,159 size 200x18; Text 'Контроль фізичної заміни енкодера / Калібровка механізму'
   Circle "Circle_27" at 262,360 size 16x16
      Appearance <- "HMI_DB_Calibration_Crane_Diagnostics_EncoderDifferenceOK"
   TextField "Text field_30" at 290,359 size 335x18; Text 'Контроль фізичної заміни енкодера / Розбіжності даних на енкодерах моста'

screen "10_ГоловнийЕкран" 800x454, template "Template_1"
   on GenerateScreen: SetTag("Tag_ScreenNumber", 10)
   TextField "Text field_1" at 69,16 size 157x21; Text 'Механізм підйому: / Механізм підйому'
   TextField "Text field_3" at 43,44 size 80x18; Text 'Швидкість'
   TextField "Text field_4" at 43,59 size 109x18; Text 'Завантаження'
   TextField "Text field_5" at 43,74 size 128x18; Text 'Координати мех.'
   IOField "I/O field_1" at 170,43 size 110x20; FormatPattern s9999.99; Unit  об/хв
      ProcessValue <- "ActVelocity_Rpm"
   IOField "I/O field_2" at 170,58 size 80x20; FormatPattern s999.99; Unit  %
      ProcessValue <- "LoadPower_Pct"
   IOField "I/O field_3" at 170,73 size 100x20; FormatPattern s99999; Unit  мм
      ProcessValue <- "Position_mm"
   Circle "Circle_40" at 15,99 size 16x16
      Appearance <- "HMI_DB_Lifting_mechanism_HL_Drive_ready"
   TextField "Text field_40" at 43,98 size 250x18; Text 'Готовність до роботи'
   Circle "Circle_21" at 15,119 size 16x16
      Appearance <- "HMI_DB_Lifting_mechanism_Thermal_protection_braking_resistor"
   TextField "Text field_21" at 43,118 size 250x18; Text 'Термозахист гальмівного резистора'
   Circle "Circle_22" at 15,139 size 16x16
      Appearance <- "HMI_DB_Lifting_mechanism_Motor_temperature_protection"
   TextField "Text field_22" at 43,138 size 250x18; Text 'Термозахист двигуна'
   Circle "Circle_1" at 15,159 size 16x16
      Appearance <- "HMI_DB_Lifting_mechanism_MD_disconnected_from_drive"
   TextField "Text field_2" at 43,158 size 250x18; Text 'РП роз'єднаний з приводом'
   Circle "Circle_2" at 15,179 size 16x16
      Appearance <- "HMI_DB_Lifting_mechanism_NSP_Enable_movement"
   TextField "Text field_6" at 43,178 size 250x18; Text 'КВ. номінальної швидкості'
   Circle "Circle_14" at 15,199 size 16x16
      Appearance <- "HMI_DB_Lifting_mechanism_Loosening_ropes"
   TextField "Text field_31" at 43,198 size 250x18; Text 'Ослаблення канатів'
   Circle "Circle_15" at 15,219 size 16x16
      Appearance <- "HMI_DB_Lifting_mechanism_1YB2_WP_MPP_disconnected_from_brake"
   TextField "Text field_32" at 43,218 size 250x18; Text 'МРР роз'єднаний з гальмом'
   Group "Group" at 23,56 size 0x25
   Group "Group_1" at 17,56 size 12x25
   GraphicView "Graphic view_2" at 672,350 size 45x45; Picture "bell-grey"
   GraphicView "Graphic view_3" at 672,350 size 45x45; Picture "bell-yellow"
      Visibility <- "HMI_DB_Sensors_CMD_Bell_On"
   Circle "Circle_30" at 15,239 size 16x16
      Appearance <- "HMI_DB_Calibration_Hoist_Calibrated"
   TextField "Text field_49" at 43,238 size 250x18; Text 'МРР роз'єднаний з гальмом / Калібровка механізму'
   TextField "Text field_7" at 378,16 size 130x21; Text 'Механізм візка: / Механізм візка'
   TextField "Text field_8" at 338,44 size 80x18; Text 'Швидкість'
   IOField "I/O field_4" at 456,43 size 110x20; FormatPattern s9999.99; Unit  об/хв
      ProcessValue <- "ActVelocity_Rpm"
   TextField "Text field_9" at 338,59 size 109x18; Text 'Завантаження'
   IOField "I/O field_5" at 456,58 size 80x20; FormatPattern s999.99; Unit  %
      ProcessValue <- "LoadPower_Pct"
   TextField "Text field_10" at 338,74 size 128x18; Text 'Координати мех.'
   IOField "I/O field_6" at 456,73 size 100x20; FormatPattern s99999; Unit  мм
      ProcessValue <- "Position_mm"
   TextField "Text field_15" at 338,98 size 250x18; Text 'Готовність до роботи'
   Circle "Circle_7" at 310,99 size 16x16
      Appearance <- "HMI_DB_Trolley_movement_mechanism_HL_Drive_ready"
   Circle "Circle_3" at 310,119 size 16x16
      Appearance <- "HMI_DB_Trolley_movement_mechanism_Engine_temperature_protection"
   TextField "Text field_11" at 338,118 size 250x18; Text 'Термозахист гальмівного резистора'
   TextField "Text field_12" at 338,138 size 250x18; Text 'Термозахист двигуна'
   Circle "Circle_4" at 310,139 size 16x16
      Appearance <- "HMI_DB_Trolley_movement_mechanism_Motor_temperature_protection"
   Circle "Circle_5" at 310,179 size 16x16
      Appearance <- "HMI_DB_Trolley_movement_mechanism_NSP_Enable_movement"
   TextField "Text field_13" at 338,178 size 250x18; Text 'КВ. номінальної швидкості'
   Circle "Circle_6" at 310,159 size 16x16
      Appearance <- "HMI_DB_Trolley_movement_mechanism_MD_disconnected_from_drive"
   TextField "Text field_14" at 338,158 size 250x18; Text 'РП роз'єднаний з приводом'
   TextField "Text field_35" at 631,43 size 160x18; Text 'Лін. конт. увімкнено'
   Circle "Circle_13" at 603,44 size 16x16
      Appearance <- "HMI_DB_PSM_HL_Line_contactor_On"
   TextField "Text field_36" at 631,63 size 160x18; Text 'Команда на увімкнення'
   Circle "Circle_16" at 603,64 size 16x16
      Appearance <- "HMI_DB_PSM_ID_Line_contactor_from_remote_control_On"
   TextField "Text field_37" at 631,83 size 160x18; Text 'Контроль напруги'
   Circle "Circle_17" at 603,84 size 16x16
      Appearance <- "HMI_DB_PSM_Input_voltage_control_380V_On"
   TextField "Text field_38" at 631,103 size 160x18; Text 'Перевант. ном. вант.'
   Circle "Circle_18" at 603,104 size 16x16
      Appearance <- "HMI_DB_Lifting_mechanism_Exceeding_rated_load_115%"
   TextField "Text field_39" at 631,123 size 160x18; Text 'КВ. рух вгору'
   Circle "Circle_19" at 603,124 size 16x16
      Appearance <- "HMI_DB_Lifting_mechanism_WP_Upward_movement"
   TextField "Text field_41" at 631,143 size 160x18; Text 'КВ. рух вниз'
   Circle "Circle_20" at 603,144 size 16x16
      Appearance <- "HMI_DB_Lifting_mechanism_WP_Downward_movement"
   TextField "Text field_42" at 631,163 size 160x18; Text 'КВ. рух вперед'
   Circle "Circle_23" at 603,164 size 16x16
      Appearance <- "HMI_DB_Trolley_movement_mechanism_WP_Forward_movement"
   TextField "Text field_43" at 631,183 size 160x18; Text 'КВ. рух назад'
   Circle "Circle_24" at 603,184 size 16x16
      Appearance <- "HMI_DB_Trolley_movement_mechanism_WP_Backward_movement"
   TextField "Text field_44" at 631,203 size 160x18; Text 'КВ. рух вліво'
   Circle "Circle_25" at 603,204 size 16x16
      Appearance <- "HMI_DB_Crane_movement_mechanism_WP_Left_movement"
   TextField "Text field_45" at 631,223 size 160x18; Text 'КВ. рух вправо'
   Circle "Circle_26" at 603,224 size 16x16
      Appearance <- "HMI_DB_Crane_movement_mechanism_WP_Right_movement"
   TextField "Text field_46" at 631,243 size 160x18; Text 'КВ. колона'
   Circle "Circle_27" at 603,244 size 16x16
      Appearance <- "HMI_DB_PSM_ColumnEnable"
   TextField "Text field_47" at 631,263 size 160x18; Text 'Сейсмодатчик'
   Circle "Circle_28" at 603,264 size 16x16
      Appearance <- "HMI_DB_Sensors_Seismic_sensor"
   TextField "Text field_48" at 631,283 size 160x18; Text 'Підігрів шаф'
   Circle "Circle_29" at 603,284 size 16x16
      Appearance <- "HMI_DB_Sensors_Cabinet_heating_control_SU1"
   Group "Group_3" at 318,56 size 0x25
   Group "Group_4" at 312,56 size 12x25
   Circle "Circle_31" at 310,199 size 16x16
      Appearance <- "HMI_DB_Calibration_Trolley_Calibrated"
   TextField "Text field_50" at 338,198 size 250x18; Text 'КВ. номінальної швидкості / Калібровка механізму'
   TextField "Text field_52" at 631,303 size 160x18; Text 'Пожежна небезпека'
   Circle "Circle_33" at 603,304 size 16x16
      Appearance <- "HMI_DB_FireAlarm_Active"
   Line "Line_11" at 23,56 size 0x25
      Visibility <- "HMI_DB_Lifting_mechanism_FirstSpeedUp"
   Line "Line_1" at 23,56 size 0x25
      Visibility <- "HMI_DB_Lifting_mechanism_FirstSpeedDown"
   Line "Line_2" at 318,56 size 0x25
      Visibility <- "HMI_DB_Trolley_movement_mechanism_FirstSpeedBackward"
   Line "Line_3" at 318,56 size 0x25
      Visibility <- "HMI_DB_Trolley_movement_mechanism_FirstSpeedForward"
   Circle "Circle_8" at 15,280 size 16x16
      Appearance <- "HMI_DB_Crane_movement_mechanism_HL_Drive_ready"
   TextField "Text field_20" at 43,279 size 250x18; Text 'Готовність до роботи'
   Circle "Circle_10" at 15,300 size 16x16
      Appearance <- "HMI_DB_Crane_movement_mechanism_NSP_Enable_movement"
   TextField "Text field_27" at 43,299 size 250x18; Text 'КВ. номінальної швидкості'
   Circle "Circle_11" at 15,320 size 16x16
      Appearance <- "HMI_DB_Crane_movement_mechanism_BreakThermalProtection"
   TextField "Text field_28" at 43,319 size 250x18; Text 'Термозахист гальмівних резисторів'
   Circle "Circle_9" at 15,340 size 16x16
      Appearance <- "HMI_DB_Crane_movement_mechanism_MotorThermalProtection"
   TextField "Text field_26" at 43,339 size 250x18; Text 'Термозахист двигунів'
   Circle "Circle_12" at 15,360 size 16x16
      Appearance <- "HMI_DB_Trolley_movement_mechanism_MD_disconnected_from_drive"
   TextField "Text field_29" at 43,359 size 250x18; Text 'РП роз'єднаний з приводом'
   TextField "Text field_16" at 283,278 size 137x21; Text 'Механізм крану: / Механізм крану'
   TextField "Text field_17" at 283,330 size 105x18; Text 'Швидкість'
   IOField "I/O field_7" at 397,329 size 75x20; FormatPattern s9999.99
      ProcessValue <- "ActVelocity_Rpm"
   TextField "Text field_18" at 283,345 size 105x18; Text 'Завантаження 4UZ1 / Завантаження'
   IOField "I/O field_8" at 397,344 size 75x20; FormatPattern s999.99
      ProcessValue <- "LoadPower_Pct"
   TextField "Text field_19" at 283,360 size 115x18; Text 'Координати мех.'
   IOField "I/O field_9" at 397,359 size 75x20; FormatPattern s99999
      ProcessValue <- "Position_mm"
   IOField "I/O field_10" at 470,329 size 110x20; FormatPattern s9999.99
      ProcessValue <- "ActVelocity_Rpm"
   IOField "I/O field_11" at 470,344 size 80x20; FormatPattern s999.99
      ProcessValue <- "LoadPower_Pct"
   IOField "I/O field_12" at 470,359 size 100x20; FormatPattern s99999
      ProcessValue <- "Position_mm"
   TextField "Text field_23" at 397,306 size 75x18; Text '4М1'
   TextField "Text field_24" at 469,306 size 75x18; Text '4М2'
   TextField "Text field_25" at 541,330 size 50x18; Text 'об/хв'
   TextField "Text field_30" at 541,345 size 50x18; Text '%'
   TextField "Text field_33" at 541,360 size 50x18; Text 'мм'
   Group "Group_2" at 455,289 size 25x0
   Group "Group_7" at 455,283 size 25x12
   Circle "Circle_32" at 15,380 size 16x16
      Appearance <- "HMI_DB_Calibration_Crane_Calibrated"
   TextField "Text field_51" at 43,379 size 250x18; Text 'РП роз'єднаний з приводом / Калібровка механізму'
   Line "Line_4" at 455,289 size 25x0
      Visibility <- "HMI_DB_Crane_movement_mechanism_FirstSpeedRight"
   Line "Line_5" at 455,289 size 25x0
      Visibility <- "HMI_DB_Crane_movement_mechanism_FirstSpeedLeft"
   TextField "Text field_34" at 614,16 size 163x21; Text 'Лінійний контактор'
   Line "Line_9" at 17,56 size 0x25
      Visibility <- "HMI_DB_Lifting_mechanism_SecondSpeedDown"
   Line "Line_8" at 17,56 size 0x25
      Visibility <- "HMI_DB_Lifting_mechanism_SecondSpeedUp"
   Line "Line_13" at 29,56 size 0x25
      Visibility <- "HMI_DB_Lifting_mechanism_SecondSpeedDown"
   Line "Line_14" at 29,56 size 0x25
      Visibility <- "HMI_DB_Lifting_mechanism_SecondSpeedUp"
   Line "Line_10" at 312,56 size 0x25
      Visibility <- "HMI_DB_Trolley_movement_mechanism_SecondSpeedBackward"
   Line "Line_12" at 324,56 size 0x25
      Visibility <- "HMI_DB_Trolley_movement_mechanism_SecondSpeedForwrd"
   Line "Line_15" at 324,56 size 0x25
      Visibility <- "HMI_DB_Trolley_movement_mechanism_SecondSpeedBackward"
   Line "Line_16" at 312,56 size 0x25
      Visibility <- "HMI_DB_Trolley_movement_mechanism_SecondSpeedForwrd"
   Line "Line_17" at 455,295 size 25x0
      Visibility <- "HMI_DB_Crane_movement_mechanism_SecondSpeedRight"
   Line "Line_18" at 455,295 size 25x0
      Visibility <- "HMI_DB_Crane_movement_mechanism_SecondSpeedLeft"
   Group "Group_5" at 455,295 size 25x0
   Group "Group_6" at 455,283 size 25x0
   Line "Line_19" at 455,283 size 25x0
      Visibility <- "HMI_DB_Crane_movement_mechanism_SecondSpeedRight"
   Line "Line_20" at 455,283 size 25x0
      Visibility <- "HMI_DB_Crane_movement_mechanism_SecondSpeedLeft"

screen "20_Механізми" 800x454, template "Template_1"
   on GenerateScreen: SetTag("Tag_ScreenNumber", 20); SetTag("iVisibilityDevices", 0)
   Circle "Circle_1" at 118,31 size 16x16
      Appearance <- "HMI_DB_PSM_Power_switch_6KV_380V_On"
      Visibility <- "iVisibilityDevices"
   TextField "Text field_1" at 146,30 size 250x18; Text '6SF1 Вимикач живлення 6KV'
      Visibility <- "iVisibilityDevices"
   Circle "Circle_2" at 118,55 size 16x16
      Appearance <- "HMI_DB_PSM_Input_voltage_control_380V_On"
      Visibility <- "iVisibilityDevices"
   TextField "Text field_2" at 146,54 size 250x18; Text '6KV Контроль напруги введення'
      Visibility <- "iVisibilityDevices"
   Circle "Circle_3" at 118,79 size 16x16
      Appearance <- "HMI_DB_PSM_Heating_circuit_breaker_220V_On"
      Visibility <- "iVisibilityDevices"
   TextField "Text field_3" at 146,78 size 250x18; Text '6SF5 Вимикач кіл живлення обігріву'
      Visibility <- "iVisibilityDevices"
   Circle "Circle_4" at 118,103 size 16x16
      Appearance <- "HMI_DB_PSM_Brake_protection_On"
      Visibility <- "iVisibilityDevices"
   TextField "Text field_4" at 146,102 size 250x18; Text '6QF2 Захист кіл гальм'
      Visibility <- "iVisibilityDevices"
   Circle "Circle_5" at 118,127 size 16x16
      Appearance <- "HMI_DB_PSM_Transformer_6T1_380V_On"
      Visibility <- "iVisibilityDevices"
   TextField "Text field_5" at 146,126 size 250x18; Text '6QF3 Вимикач трансформатора 6T1'
      Visibility <- "iVisibilityDevices"
   Circle "Circle_6" at 420,151 size 16x16
      Appearance <- "HMI_DB_PSM_Transformer_sec_circuit_breaker_6T1_380V_On"
      Visibility <- "iVisibilityDevices"
   TextField "Text field_6" at 448,150 size 345x18; Text '6QF4 Вимикач втор. кіл трансформатора 6T1'
      Visibility <- "iVisibilityDevices"
   Circle "Circle_7" at 118,175 size 16x16
      Appearance <- "HMI_DB_PSM_ID_Control_circuit_breaker_220V_On"
      Visibility <- "iVisibilityDevices"
   TextField "Text field_7" at 146,174 size 250x18; Text '6SF2 Вимикач кіл управління 220в'
      Visibility <- "iVisibilityDevices"
   Circle "Circle_8" at 118,199 size 16x16
      Appearance <- "HMI_DB_PSM_ID_ORP_power_circuit_breaker_220V_On"
      Visibility <- "iVisibilityDevices"
   TextField "Text field_8" at 146,198 size 250x18; Text '6SF4 Вимикач кіл живлення ОВП'
      Visibility <- "iVisibilityDevices"
   Circle "Circle_9" at 118,223 size 16x16
      Appearance <- "HMI_DB_PSM_Cabinet_circuit_breaker_220V_On"
      Visibility <- "iVisibilityDevices"
   TextField "Text field_9" at 146,222 size 250x18; Text '9QF4 Вимикач власних потреб шафи'
      Visibility <- "iVisibilityDevices"
   Circle "Circle_10" at 118,247 size 16x16
      Appearance <- "HMI_DB_Sensors_Cabinet_heating_control_SU1"
      Visibility <- "iVisibilityDevices"
   TextField "Text field_10" at 146,246 size 250x18; Text '9K2 Контроль підігріву шафи'
      Visibility <- "iVisibilityDevices"
   Circle "Circle_11" at 118,271 size 16x16
      Appearance <- "HMI_DB_Lifting_mechanism_1YB1_Brake_rectifier_protection"
      Visibility <- "iVisibilityDevices"
   TextField "Text field_11" at 146,270 size 250x18; Text '1QF1 Захист випрямляча гальма 1YB1'
      Visibility <- "iVisibilityDevices"
   Circle "Circle_12" at 118,295 size 16x16
      Appearance <- "HMI_DB_Lifting_mechanism_1YB2_Brake_rectifier_protection"
      Visibility <- "iVisibilityDevices"
   TextField "Text field_12" at 146,294 size 250x18; Text '1QF2 Захист випрямляча гальма 1YB2'
      Visibility <- "iVisibilityDevices"
   Circle "Circle_13" at 118,319 size 16x16
      Appearance <- "HMI_DB_Crane_movement_mechanism_Brake_protection_On"
      Visibility <- "iVisibilityDevices"
   TextField "Text field_13" at 146,318 size 250x18; Text '4QF1 Захист кіл гальм'
      Visibility <- "iVisibilityDevices"
   Circle "Circle_14" at 420,271 size 16x16
      Appearance <- "HMI_DB_Lifting_mechanism_1YB2_WP_MPP_disconnected_from_brake"
      Visibility <- "iVisibilityDevices"
   TextField "Text field_14" at 448,270 size 345x18; Text '1SQ33 Гальмо 1YB2 дозв. роб. (МРР роз'єд. з гальм)'
      Visibility <- "iVisibilityDevices"
   Circle "Circle_15" at 420,295 size 16x16
      Appearance <- "HMI_DB_Lifting_mechanism_MD_disconnected_from_drive"
      Visibility <- "iVisibilityDevices"
   TextField "Text field_15" at 448,294 size 345x18; Text '1SQ41 Дозвіл роботи мех. підйому, ручн. привід'
      Visibility <- "iVisibilityDevices"
   Circle "Circle_16" at 420,31 size 16x16
      Appearance <- "HMI_DB_Trolley_movement_mechanism_MD_disconnected_from_drive"
      Visibility <- "iVisibilityDevices"
   TextField "Text field_16" at 448,30 size 345x18; Text '3SQ41 Дозвіл роботи - РП роз'єд. з привод.'
      Visibility <- "iVisibilityDevices"
   Circle "Circle_17" at 420,55 size 16x16
      Appearance <- "HMI_DB_Crane_movement_mechanism_4SQ41_MD_disconnected_from_drive"
      Visibility <- "iVisibilityDevices"
   TextField "Text field_17" at 448,54 size 345x18; Text '4SQ41 Дозвіл роботи - РП роз'єд. з привод.'
      Visibility <- "iVisibilityDevices"
   Circle "Circle_18" at 420,79 size 16x16
      Appearance <- "HMI_DB_Crane_movement_mechanism_4SQ42_MD_disconnected_from_drive"
      Visibility <- "iVisibilityDevices"
   TextField "Text field_18" at 448,78 size 345x18; Text '4SQ42 Дозвіл роботи - РП роз'єд. з привод.'
      Visibility <- "iVisibilityDevices"
   Circle "Circle_19" at 420,103 size 16x16
      Appearance <- "HMI_DB_Crane_movement_mechanism_WP_Right_movement"
      Visibility <- "iVisibilityDevices"
   TextField "Text field_19" at 448,102 size 345x18; Text '4SQ2.2 Дозвіл роботи моста, рух вправо'
      Visibility <- "iVisibilityDevices"
   Circle "Circle_20" at 420,127 size 16x16
      Appearance <- "HMI_DB_Crane_movement_mechanism_WP_Left_movement"
      Visibility <- "iVisibilityDevices"
   TextField "Text field_20" at 448,126 size 345x18; Text '4SQ2.1 Дозвіл роботи моста, рух вліво'
      Visibility <- "iVisibilityDevices"
   Circle "Circle_21" at 420,175 size 16x16
      Appearance <- "HMI_DB_Lifting_mechanism_WP_Downward_movement"
      Visibility <- "iVisibilityDevices"
   TextField "Text field_21" at 448,174 size 345x18; Text '1SQ1.4 Дозвіл роботи підйому, рух вниз'
      Visibility <- "iVisibilityDevices"
   Circle "Circle_22" at 420,199 size 16x16
      Appearance <- "HMI_DB_Lifting_mechanism_WP_Upward_movement"
      Visibility <- "iVisibilityDevices"
   TextField "Text field_22" at 448,198 size 345x18; Text '1SQ1.3 Дозвіл роботи підйому, pух вгору'
      Visibility <- "iVisibilityDevices"
   Circle "Circle_23" at 420,223 size 16x16
      Appearance <- "HMI_DB_Trolley_movement_mechanism_WP_Backward_movement"
      Visibility <- "iVisibilityDevices"
   TextField "Text field_23" at 448,222 size 345x18; Text '3SQ2.2 Дозвіл роботи візка, рух назад'
      Visibility <- "iVisibilityDevices"
   Circle "Circle_24" at 420,247 size 16x16
      Appearance <- "HMI_DB_Trolley_movement_mechanism_WP_Forward_movement"
      Visibility <- "iVisibilityDevices"
   TextField "Text field_24" at 448,246 size 345x18; Text '3SQ1.2 Дозвіл роботи візка, рух вперед'
      Appearance <- "HMI_DB_Trolley_movement_mechanism_WP_Forward_movement"
      Visibility <- "iVisibilityDevices"
   Circle "Circle_25" at 118,151 size 16x16
      Appearance <- "HMI_DB_Sensors_Seismic_sensor"
      Visibility <- "iVisibilityDevices"
   TextField "Text field_25" at 146,150 size 250x18; Text '9K3 Сейсмодатчик'
      Visibility <- "iVisibilityDevices"
   Circle "Circle_26" at 118,343 size 16x16
      Visibility <- "iVisibilityDevices"
      Appearance <- "Data_base_Profinet_Ok"
   TextField "Text field_26" at 146,342 size 250x18; Text 'Комунікація профінет'
      Visibility <- "iVisibilityDevices"
   Circle "Circle_27" at 420,343 size 16x16
      Visibility <- "iVisibilityDevices"
      Appearance <- "HMI_DB_PSM_Zero_Protection"
   TextField "Text field_27" at 448,342 size 250x18; Text 'Нульове блокування'
      Visibility <- "iVisibilityDevices"
   Circle "Circle_48" at 420,319 size 16x16
      Visibility <- "iVisibilityDevices"
      Appearance <- "HMI_DB_PSM_ID_Line_contactor_from_remote_control_On"
   TextField "Text field_48" at 448,318 size 345x18; Text '6KM1 Лінійний контактор увімкнений'
      Visibility <- "iVisibilityDevices"
   Circle "Circle_49" at 118,7 size 16x16
      Visibility <- "iVisibilityDevices"
      Appearance <- "HMI_DB_PSM_ID_Line_contactor_from_remote_control_On"
   TextField "Text field_49" at 146,6 size 250x18; Text 'Команда на увімк. голов. контактору / Головний контактор увімкнено'
      Visibility <- "iVisibilityDevices"
   Circle "Circle_54" at 420,7 size 16x16
      Visibility <- "iVisibilityDevices"
      Appearance <- "HMI_DB_PSM_Control_contactor_220V_On"
   TextField "Text field_54" at 448,6 size 345x18; Text '6KM2 Контактор кіл керування 220В увімкнен.'
      Visibility <- "iVisibilityDevices"
   TextField "Text field_63" at 146,366 size 250x18; Text '1K11 Перевант. ном. вант.'
      Visibility <- "iVisibilityDevices"
   Circle "Circle_61" at 118,367 size 16x16
      Appearance <- "HMI_DB_Lifting_mechanism_Exceeding_rated_load_115%"
      Visibility <- "iVisibilityDevices"
   TextField "Text field_64" at 448,366 size 350x18; Text '4К5, 3К3 Дозвіл роб. з будь якої сторони від колони'
      Visibility <- "iVisibilityDevices"
   Circle "Circle_62" at 420,367 size 16x16
      Appearance <- "HMI_DB_PSM_ColumnEnable"
      Visibility <- "iVisibilityDevices"
   TextField "Text field_68" at 146,390 size 250x18; Text 'Пожежна небезпека'
      Visibility <- "iVisibilityDevices"
   Circle "Circle_65" at 118,391 size 16x16
      Visibility <- "iVisibilityDevices"
      Appearance <- "HMI_DB_FireAlarm_Active"
   Button "btnLiftUp" at 8,120 size 96x32; TextOff 'Механізм підйому'
      on Release: SetTag("iVisibilityDevices", 1)
      Appearance <- "iVisibilityDevices"
   Button "btnTrolley" at 8,160 size 96x32; TextOff 'Механізм візка'
      on Click: SetTag("iVisibilityDevices", 2)
      Appearance <- "iVisibilityDevices"
   Button "btnCrane" at 8,200 size 96x32; TextOff 'Механізм крану'
      on Release: SetTag("iVisibilityDevices", 3)
      Appearance <- "iVisibilityDevices"
   Button "btnContactor" at 8,80 size 96x32; TextOff 'Лінійний контактор'
      on Release: SetTag("iVisibilityDevices", 0)
      Appearance <- "iVisibilityDevices"
   Button "btnCrane_1" at 8,240 size 96x32; TextOff 'Власні потреби'
      on Release: SetTag("iVisibilityDevices", 4)
      Appearance <- "iVisibilityDevices"
   Circle "Circle_28" at 119,103 size 16x16
      Appearance <- "HMI_DB_PSM_CMD_Line_contactor_Off"
      Visibility <- "iVisibilityDevices"
   TextField "Text field_28" at 147,102 size 270x18; Text 'Головний контактор увімкнено'
      Visibility <- "iVisibilityDevices"
   Circle "Circle_29" at 420,103 size 16x16
      Appearance <- "HMI_DB_Lifting_mechanism_Thermal_protection_braking_resistor"
      Visibility <- "iVisibilityDevices"
   TextField "Text field_29" at 448,102 size 290x18; Text '1BT1 Термозахист гальмівного резистора'
      Visibility <- "iVisibilityDevices"
   Circle "Circle_30" at 420,127 size 16x16
      Appearance <- "HMI_DB_Lifting_mechanism_Motor_temperature_protection"
      Visibility <- "iVisibilityDevices"
   TextField "Text field_30" at 448,126 size 250x18; Text '1KT Термозахист двигуна'
      Visibility <- "iVisibilityDevices"
   Circle "Circle_31" at 420,151 size 16x16
      Appearance <- "HMI_DB_Lifting_mechanism_1YB1_Thickness_brake_pads_normal"
      Visibility <- "iVisibilityDevices"
   TextField "Text field_31" at 448,150 size 290x18; Text '1SQ23 Товщина гальмівних накладок 1MB1'
      Visibility <- "iVisibilityDevices"
   Circle "Circle_32" at 420,175 size 16x16
      Appearance <- "HMI_DB_Lifting_mechanism_Brake_wear_control"
      Visibility <- "iVisibilityDevices"
   TextField "Text field_32" at 448,174 size 310x18; Text '1BM1-6k Контроль зносу гальма мех. підйому'
      Visibility <- "iVisibilityDevices"
   Circle "Circle_33" at 420,199 size 16x16
      Appearance <- "HMI_DB_Lifting_mechanism_Loosening_ropes"
      Visibility <- "iVisibilityDevices"
   TextField "Text field_33" at 448,198 size 310x18; Text '1K12 Ослаблення канатів'
      Visibility <- "iVisibilityDevices"
   Circle "Circle_50" at 420,247 size 16x16
      Visibility <- "iVisibilityDevices"
      Appearance <- "HMI_DB_Calibration_Hoist_Calibrated"
   TextField "Text field_50" at 448,246 size 310x18; Text 'Калібровка механізму'
      Visibility <- "iVisibilityDevices"
   Circle "Circle_53" at 420,223 size 16x16
      Visibility <- "iVisibilityDevices"
      Appearance <- "HMI_DB_Lifting_mechanism_Exceeding_rated_load_115%"
   TextField "Text field_53" at 448,222 size 310x18; Text '1K11 Перевищення номінального вантажу'
      Visibility <- "iVisibilityDevices"
   TextField "Text field_55" at 119,362 size 121x21; Text 'Статус роботи'
      Visibility <- "iVisibilityDevices"
   SymbolicIOField "Symbolic I/O field_3" at 294,357 size 480x32; TextOff '0'; TextOn '1'; TextList "LiftUpStatus"
      Visibility <- "iVisibilityDevices"
      ProcessValue <- "HMI_DB_Lifting_mechanism_LM_Status"
   Circle "Circle_55" at 119,127 size 16x16
      Visibility <- "iVisibilityDevices"
      Appearance <- "HMI_DB_Sensors_Drum_rotation_control"
   TextField "Text field_56" at 147,126 size 270x18; Text '1BV Контроль обертання барабану'
      Visibility <- "iVisibilityDevices"
   Circle "Circle_56" at 119,271 size 16x16
      Visibility <- "iVisibilityDevices"
      Appearance <- "HMI_DB_Lifting_mechanism_Work_control"
   TextField "Text field_58" at 147,270 size 270x18; Text '1BМ1 Контроль роботи мех. підйому'
      Visibility <- "iVisibilityDevices"
   Circle "Circle_57" at 119,151 size 16x16
      Visibility <- "iVisibilityDevices"
      Appearance <- "HMI_DB_Lifting_mechanism_1YB1_Brake released"
   TextField "Text field_59" at 147,150 size 270x18; Text '1SQ21 Гальмо розгальмоване (1МВ1)'
      Visibility <- "iVisibilityDevices"
   Circle "Circle_58" at 119,175 size 16x16
      Visibility <- "iVisibilityDevices"
      Appearance <- "HMI_DB_Lifting_mechanism_1YB1_Brake_applied"
   TextField "Text field_60" at 147,174 size 270x18; Text '1SQ22 Гальмо загальмоване (1МВ1)'
      Visibility <- "iVisibilityDevices"
   Circle "Circle_59" at 119,199 size 16x16
      Visibility <- "iVisibilityDevices"
      Appearance <- "HMI_DB_Lifting_mechanism_1YB2_Brake released"
   TextField "Text field_61" at 147,198 size 270x18; Text '1SQ31.1 Гальмо розгальмоване (1YВ2)'
      Visibility <- "iVisibilityDevices"
   Circle "Circle_60" at 119,223 size 16x16
      Visibility <- "iVisibilityDevices"
      Appearance <- "HMI_DB_Lifting_mechanism_1YB2_Brake_applied"
   TextField "Text field_62" at 147,222 size 270x18; Text '1SQ31.2 Гальмо загальмоване (1YВ2)'
      Visibility <- "iVisibilityDevices"
   Circle "Circle_34" at 119,247 size 16x16
      Visibility <- "iVisibilityDevices"
      Appearance <- "Error"
   TextField "Text field_34" at 147,246 size 270x18; Text '1UZ1 Помилка ПЧ'
      Visibility <- "iVisibilityDevices"
   Circle "Circle_35" at 119,103 size 16x16
      Appearance <- "HMI_DB_PSM_CMD_Line_contactor_Off"
      Visibility <- "iVisibilityDevices"
   TextField "Text field_35" at 147,102 size 310x18; Text 'Головний контактор увімкнено'
      Visibility <- "iVisibilityDevices"
   Circle "Circle_36" at 119,127 size 16x16
      Appearance <- "HMI_DB_Lifting_mechanism_Exceeding_rated_load_115%"
      Visibility <- "iVisibilityDevices"
   TextField "Text field_36" at 147,126 size 320x18; Text '1K11 Перевищення номінального вантажу'
      Visibility <- "iVisibilityDevices"
   Circle "Circle_37" at 119,151 size 16x16
      Appearance <- "HMI_DB_Trolley_movement_mechanism_Engine_temperature_protection"
      Visibility <- "iVisibilityDevices"
   TextField "Text field_37" at 147,150 size 310x18; Text '3BT1 Термозахист гальмівного резистора'
      Visibility <- "iVisibilityDevices"
   Circle "Circle_38" at 119,175 size 16x16
      Appearance <- "HMI_DB_Trolley_movement_mechanism_Motor_temperature_protection"
      Visibility <- "iVisibilityDevices"
   TextField "Text field_38" at 147,174 size 310x18; Text '3KT Термозахист двигуна'
      Visibility <- "iVisibilityDevices"
   Circle "Circle_39" at 119,223 size 16x16
      Visibility <- "iVisibilityDevices"
      Appearance <- "Error"
   TextField "Text field_39" at 147,222 size 310x18; Text '3UZ1 Помилка ПЧ'
      Visibility <- "iVisibilityDevices"
   Circle "Circle_51" at 119,199 size 16x16
      Visibility <- "iVisibilityDevices"
      Appearance <- "HMI_DB_Calibration_Trolley_Calibrated"
   TextField "Text field_51" at 147,198 size 310x18; Text 'Калібровка механізму'
      Visibility <- "iVisibilityDevices"
   TextField "Text field_57" at 119,362 size 121x21; Text 'Статус роботи'
      Visibility <- "iVisibilityDevices"
   SymbolicIOField "Symbolic I/O field_1" at 294,357 size 480x32; TextOff '0'; TextOn '1'; TextList "TrolleyStatus"
      Visibility <- "iVisibilityDevices"
      ProcessValue <- "HMI_DB_Trolley_movement_mechanism_TM_Status"
   Circle "Circle_40" at 119,103 size 16x16
      Appearance <- "HMI_DB_PSM_CMD_Line_contactor_Off"
      Visibility <- "iVisibilityDevices"
   TextField "Text field_40" at 147,102 size 290x18; Text 'Головний контактор увімкнено'
      Visibility <- "iVisibilityDevices"
   Circle "Circle_41" at 119,127 size 16x16
      Appearance <- "HMI_DB_Lifting_mechanism_Exceeding_rated_load_115%"
      Visibility <- "iVisibilityDevices"
   TextField "Text field_41" at 147,126 size 320x18; Text '1K11 Перевищення номінального вантажу'
      Visibility <- "iVisibilityDevices"
   Circle "Circle_42" at 119,151 size 16x16
      Appearance <- "HMI_DB_Crane_movement_mechanism_4RT1_thermal_protection_braking_resistor"
      Visibility <- "iVisibilityDevices"
   TextField "Text field_42" at 147,150 size 300x18; Text '4BT1 Термозахист гальмівного резистора'
      Visibility <- "iVisibilityDevices"
   Circle "Circle_43" at 119,175 size 16x16
      Appearance <- "HMI_DB_Crane_movement_mechanism_4RT2_thermal_protection_braking_resistor"
      Visibility <- "iVisibilityDevices"
   TextField "Text field_43" at 147,174 size 300x18; Text '4BT2 Термозахист гальмівного резистора'
      Visibility <- "iVisibilityDevices"
   Circle "Circle_44" at 119,199 size 16x16
      Appearance <- "HMI_DB_Crane_movement_mechanism_4M1_engine_temperature_protection"
      Visibility <- "iVisibilityDevices"
   TextField "Text field_44" at 147,198 size 290x18; Text '4KT1 Термозахист двигуна 4М1'
      Visibility <- "iVisibilityDevices"
   Circle "Circle_45" at 119,223 size 16x16
      Appearance <- "HMI_DB_Crane_movement_mechanism_4M2_engine_temperature_protection"
      Visibility <- "iVisibilityDevices"
   TextField "Text field_45" at 147,222 size 290x18; Text '4KT2 Термозахист двигуна 4М2'
      Visibility <- "iVisibilityDevices"
   Circle "Circle_46" at 119,271 size 16x16
      Visibility <- "iVisibilityDevices"
      Appearance <- "Error"
   TextField "Text field_46" at 147,270 size 290x18; Text '4UZ1 Помилка ПЧ'
      Visibility <- "iVisibilityDevices"
   Circle "Circle_47" at 119,295 size 16x16
      Visibility <- "iVisibilityDevices"
      Appearance <- "Error"
   TextField "Text field_47" at 147,294 size 290x18; Text '4UZ2 Помилка ПЧ'
      Visibility <- "iVisibilityDevices"
   Circle "Circle_52" at 119,247 size 16x16
      Visibility <- "iVisibilityDevices"
      Appearance <- "HMI_DB_Calibration_Crane_Calibrated"
   TextField "Text field_52" at 147,246 size 290x18; Text 'Калібровка'
      Visibility <- "iVisibilityDevices"
   TextField "Text field_67" at 119,362 size 121x21; Text 'Статус роботи'
      Visibility <- "iVisibilityDevices"
   SymbolicIOField "Symbolic I/O field_2" at 294,357 size 480x32; TextOff '0'; TextOn '1'; TextList "CraneStatus"
      Visibility <- "iVisibilityDevices"
      ProcessValue <- "HMI_DB_Crane_movement_mechanism_CM_Status"
   Circle "Circle_63" at 119,103 size 16x16
      Visibility <- "iVisibilityDevices"
      Appearance <- "HMI_DB_PSM_Transformer_9T1_380V_On"
   TextField "Text field_65" at 147,102 size 290x18; Text '9QF2 Вимикач транформатора 9Т1, 380в'
      Visibility <- "iVisibilityDevices"
   Circle "Circle_64" at 119,127 size 16x16
      Visibility <- "iVisibilityDevices"
      Appearance <- "HMI_DB_PSM_Repair_lighting_switch_12V_On"
   TextField "Text field_66" at 147,126 size 320x18; Text '9QF3 Вимикач ремонтного освітлення 12В'
      Visibility <- "iVisibilityDevices"

screen "81_КалібровкаПідйому" 800x454, template "Template_1"
   on GenerateScreen: SetTag("Tag_ScreenNumber", 81)
   IOField "I/O field_3" at 365,32 size 70x25; FormatPattern 99999
      ProcessValue <- "HMI_DB_Calibration_Hoist_CurrentStep"
   IOField "I/O field_4" at 365,32 size 70x25; FormatPattern 99999
      ProcessValue <- "HMI_DB_Calibration_Hoist_CurrentStep"
      Visibility <- "HMI_DB_Calibration_Hoist_Calibrated"
   IOField "I/O field_5" at 365,32 size 70x25; FormatPattern 99999
      ProcessValue <- "HMI_DB_Calibration_Hoist_CurrentStep"
      Visibility <- "HMI_DB_Calibration_Hoist_Active"
   IOField "I/O field_6" at 365,32 size 70x25; FormatPattern 99999
      ProcessValue <- "HMI_DB_Calibration_Hoist_CurrentStep"
      Visibility <- "HMI_DB_Calibration_Hoist_Aborted"
   IOField "I/O field_7" at 365,32 size 70x25; FormatPattern 99999
      ProcessValue <- "HMI_DB_Calibration_Hoist_CurrentStep"
      Visibility <- "HMI_DB_Calibration_Hoist_Fault"
   TextField "Text field_12" at 681,263 size 30x18; Text '110'
   TextField "Text field_13" at 23,263 size 22x18; Text '10'
   TextField "Text field_14" at 89,263 size 22x18; Text '20'
   TextField "Text field_15" at 155,263 size 22x18; Text '30'
   TextField "Text field_16" at 221,263 size 22x18; Text '40'
   TextField "Text field_17" at 288,263 size 22x18; Text '50'
   TextField "Text field_18" at 354,263 size 22x18; Text '60'
   TextField "Text field_19" at 420,263 size 22x18; Text '70'
   TextField "Text field_20" at 486,263 size 22x18; Text '80'
   TextField "Text field_21" at 553,263 size 22x18; Text '90'
   TextField "Text field_22" at 615,263 size 30x18; Text '100'
   TextField "Text field_24" at 748,263 size 30x18; Text '130'
   Circle "Circle_14" at 26,342 size 16x16
      Visibility <- "HMI_DB_Calibration_Hoist_Steps_Active_Step10"
   Circle "Circle_15" at 26,342 size 16x16
      Visibility <- "HMI_DB_Calibration_Hoist_Steps_Completed_Step10"
   Circle "Circle_17" at 92,342 size 16x16
      Visibility <- "HMI_DB_Calibration_Hoist_Steps_Active_Step20"
   Circle "Circle_18" at 92,342 size 16x16
      Visibility <- "HMI_DB_Calibration_Hoist_Steps_Completed_Step20"
   Circle "Circle_20" at 158,342 size 16x16
      Visibility <- "HMI_DB_Calibration_Hoist_Steps_Active_Step30"
   Circle "Circle_21" at 158,342 size 16x16
      Visibility <- "HMI_DB_Calibration_Hoist_Steps_Completed_Step30"
   Circle "Circle_23" at 224,342 size 16x16
      Visibility <- "HMI_DB_Calibration_Hoist_Steps_Active_Step40"
   Circle "Circle_24" at 224,342 size 16x16
      Visibility <- "HMI_DB_Calibration_Hoist_Steps_Completed_Step40"
   Circle "Circle_26" at 291,342 size 16x16
      Visibility <- "HMI_DB_Calibration_Hoist_Steps_Active_Step50"
   Circle "Circle_27" at 291,342 size 16x16
      Visibility <- "HMI_DB_Calibration_Hoist_Steps_Completed_Step50"
   Circle "Circle_29" at 357,342 size 16x16
      Visibility <- "HMI_DB_Calibration_Hoist_Steps_Active_Step60"
   Circle "Circle_30" at 357,342 size 16x16
      Visibility <- "HMI_DB_Calibration_Hoist_Steps_Completed_Step60"
   Circle "Circle_32" at 423,342 size 16x16
      Visibility <- "HMI_DB_Calibration_Hoist_Steps_Active_Step70"
   Circle "Circle_33" at 423,342 size 16x16
      Visibility <- "HMI_DB_Calibration_Hoist_Steps_Completed_Step70"
   Circle "Circle_35" at 489,342 size 16x16
      Visibility <- "HMI_DB_Calibration_Hoist_Steps_Active_Step80"
   Circle "Circle_36" at 489,342 size 16x16
      Visibility <- "HMI_DB_Calibration_Hoist_Steps_Completed_Step80"
   Circle "Circle_38" at 556,342 size 16x16
      Visibility <- "HMI_DB_Calibration_Hoist_Steps_Active_Step90"
   Circle "Circle_39" at 556,342 size 16x16
      Visibility <- "HMI_DB_Calibration_Hoist_Steps_Completed_Step90"
   Circle "Circle_41" at 622,342 size 16x16
      Visibility <- "HMI_DB_Calibration_Hoist_Steps_Active_Step100"
   Circle "Circle_42" at 622,342 size 16x16
      Visibility <- "HMI_DB_Calibration_Hoist_Steps_Completed_Step100"
   Circle "Circle_44" at 688,342 size 16x16
      Visibility <- "HMI_DB_Calibration_Hoist_Steps_Active_Step110"
   Circle "Circle_45" at 688,342 size 16x16
      Visibility <- "HMI_DB_Calibration_Hoist_Steps_Completed_Step110"
   Circle "Circle_47" at 755,342 size 16x16
      Visibility <- "HMI_DB_Calibration_Hoist_Steps_Active_Step130"
   Circle "Circle_48" at 755,342 size 16x16
      Visibility <- "HMI_DB_Calibration_Hoist_Steps_Completed_Step130"
   Line "Line_11" at 303,58 size 0x25
      Visibility <- "HMI_DB_Lifting_mechanism_FirstSpeedUp"
   Line "Line_3" at 303,58 size 0x25
      Visibility <- "HMI_DB_Lifting_mechanism_FirstSpeedDown"
   TextField "Text field_41" at 82,33 size 169x23; Text 'НЕ КАЛІБРОВАНО'
      Visibility <- "HMI_DB_Calibration_Hoist_Calibrated"
   TextField "Text field_4" at 38,33 size 258x23; Text 'КАЛІБРОВКА АНУЛЬОВАНА'
      Visibility <- "HMI_DB_Calibration_Hoist_Aborted"
   TextField "Text field_3" at 55,33 size 223x23; Text 'ПОМИЛКА КАЛІБРОВКИ'
      Visibility <- "HMI_DB_Calibration_Hoist_Fault"
   TextField "Text field_2" at 57,33 size 219x23; Text 'КАЛІБРОВКА АКТИВНА'
      Visibility <- "HMI_DB_Calibration_Hoist_Active"
   TextField "Text field_1" at 97,33 size 139x23; Text 'КАЛІБРОВАНО'
      Visibility <- "HMI_DB_Calibration_Hoist_Calibrated"
   Group "Group" at 38,33 size 258x23
   TextField "Text field_5" at 8,61 size 61x18; Text 'Позиція'
   TextField "Text field_6" at 8,85 size 136x18; Text 'Реперний вимикач'
   TextField "Text field_7" at 8,109 size 80x18; Text 'Швидкість'
   TextField "Text field_8" at 365,133 size 104x18; Text 'Залишок часу'
   IOField "I/O field_1" at 184,54 size 120x32; FormatPattern s999999; Unit  мм
      ProcessValue <- "HMI_DB_Calibration_Hoist_Position_mm"
   IOField "I/O field_2" at 184,102 size 120x32; FormatPattern s9999.99; Unit  об/хв
      ProcessValue <- "HMI_DB_Calibration_Hoist_DriveVelocity_rpm"
   Circle "Circle_49" at 236,86 size 16x16
      Appearance <- "HMI_DB_Calibration_Hoist_Reference1K1"
   TextField "Text field_9" at 34,5 size 267x21; Text 'Статус калібровки мех. підйому'
   TextField "Text field_10" at 482,5 size 181x21; Text 'Поточний крок та дія'
   Group "Group_1" at 365,32 size 70x25
   SymbolicIOField "Symbolic I/O field_1" at 453,29 size 327x32; TextOff '0'; TextOn '1'; TextList "LiftUpStepName"
      ProcessValue <- "HMI_DB_Calibration_Hoist_CurrentStep"
   TextField "Text field_11" at 365,85 size 268x18; Text 'Умови переходу на наступний крок:'
   SymbolicIOField "Symbolic I/O field_2" at 365,102 size 416x32; TextOff '0'; TextOn '1'; TextList "LiftUpCondition"
      ProcessValue <- "HMI_DB_Calibration_Hoist_CurrentStep"
   Group "Group_2" at 680,256 size 32x32
   Group "Group_3" at 18,256 size 32x32
   Group "Group_4" at 84,256 size 32x32
   Group "Group_5" at 150,256 size 32x32
   Group "Group_6" at 216,256 size 32x32
   Group "Group_7" at 283,256 size 32x32
   Group "Group_8" at 349,256 size 32x32
   Group "Group_9" at 415,256 size 32x32
   Group "Group_10" at 481,256 size 32x32
   Group "Group_11" at 548,256 size 32x32
   Group "Group_12" at 614,256 size 32x32
   Group "Group_14" at 747,256 size 32x32
   TextField "Text field_23" at 0,295 size 68x28; Text 'Перевірка умов'
   TextField "Text field_25" at 68,295 size 65x40; Text 'Натисніть кнопку "Підйом"'
   TextField "Text field_26" at 133,295 size 67x40; Text 'Рух до реперної точки 1К1'
   TextField "Text field_27" at 198,295 size 69x40; Text 'Відпустіть кнопку "Підйом"'
   TextField "Text field_28" at 263,295 size 73x40; Text 'Опускайте механізм нижче 1К1'
   TextField "Text field_29" at 330,295 size 70x28; Text 'Відхід завершено'
   TextField "Text field_30" at 399,295 size 65x40; Text 'Натисніть кнопку "Підйом"'
   TextField "Text field_31" at 462,295 size 70x40; Text 'Повторний підхід до 1К1'
   TextField "Text field_32" at 544,295 size 40x28; Text 'Quick Stop'
   TextField "Text field_33" at 593,295 size 75x40; Text 'Очікування зупинки привода'
   TextField "Text field_34" at 665,295 size 62x40; Text 'Запуск preset енкодера'
   TextField "Text field_35" at 725,295 size 75x40; Text 'Калібровку успішно завершено'
   Group "Group_13" at 26,342 size 16x16
   Group "Group_15" at 92,342 size 16x16
   Group "Group_16" at 158,342 size 16x16
   Group "Group_17" at 224,342 size 16x16
   Group "Group_18" at 291,342 size 16x16
   Group "Group_19" at 357,342 size 16x16
   Group "Group_20" at 423,342 size 16x16
   Group "Group_21" at 489,342 size 16x16
   Group "Group_22" at 556,342 size 16x16
   Group "Group_23" at 622,342 size 16x16
   Group "Group_24" at 688,342 size 16x16
   Group "Group_25" at 755,342 size 16x16
   TextField "Text field_36" at 18,381 size 148x18; Text 'Умовні позначення:'
   TextField "Text field_37" at 190,381 size 85x18; Text '- Виконано'
   TextField "Text field_38" at 365,381 size 124x18; Text '- Поточний крок'
   TextField "Text field_39" at 540,381 size 92x18; Text '- Очікується'
   TextField "Text field_40" at 205,226 size 387x21; Text 'Послідовність кроків калібровки мех. підйому'
   IOField "I/O field_8" at 541,126 size 60x32; FormatPattern 999; Unit  хв :
      ProcessValue <- "HMI_DB_Calibration_Hoist_TimerRemaining_Min"
   IOField "I/O field_9" at 595,126 size 55x32; FormatPattern 999; Unit  сек
      ProcessValue <- "HMI_DB_Calibration_Hoist_TimerRemaining_Sec"
   Group "Group_26" at 303,58 size 0x25
   TextField "Text field_42" at 8,133 size 88x18; Text 'Інкременти'
   IOField "I/O field_10" at 184,132 size 100x20; FormatPattern s9999999999
      ProcessValue <- "RawPosition"

screen "82_КалібровкаВізка" 800x454, template "Template_1"
   on GenerateScreen: SetTag("Tag_ScreenNumber", 82)
   IOField "I/O field_3" at 365,32 size 70x25; FormatPattern 99999
      ProcessValue <- "HMI_DB_Calibration_Trolley_CurrentStep"
   IOField "I/O field_4" at 365,32 size 70x25; FormatPattern 99999
      Visibility <- "HMI_DB_Calibration_Trolley_Calibrated"
      ProcessValue <- "HMI_DB_Calibration_Trolley_CurrentStep"
   IOField "I/O field_5" at 365,32 size 70x25; FormatPattern 99999
      ProcessValue <- "HMI_DB_Calibration_Trolley_CurrentStep"
      Visibility <- "HMI_DB_Calibration_Trolley_Active"
   IOField "I/O field_6" at 365,32 size 70x25; FormatPattern 99999
      ProcessValue <- "HMI_DB_Calibration_Trolley_CurrentStep"
      Visibility <- "HMI_DB_Calibration_Trolley_Aborted"
   IOField "I/O field_7" at 365,32 size 70x25; FormatPattern 99999
      ProcessValue <- "HMI_DB_Calibration_Trolley_CurrentStep"
      Visibility <- "HMI_DB_Calibration_Trolley_Fault"
   TextField "Text field_12" at 681,263 size 30x18; Text '110'
   TextField "Text field_13" at 23,263 size 22x18; Text '10'
   TextField "Text field_14" at 89,263 size 22x18; Text '20'
   TextField "Text field_15" at 155,263 size 22x18; Text '30'
   TextField "Text field_16" at 221,263 size 22x18; Text '40'
   TextField "Text field_17" at 288,263 size 22x18; Text '50'
   TextField "Text field_18" at 354,263 size 22x18; Text '60'
   TextField "Text field_19" at 420,263 size 22x18; Text '70'
   TextField "Text field_20" at 486,263 size 22x18; Text '80'
   TextField "Text field_21" at 553,263 size 22x18; Text '90'
   TextField "Text field_22" at 615,263 size 30x18; Text '100'
   TextField "Text field_24" at 748,263 size 30x18; Text '130'
   TextField "Text field_5" at 8,61 size 61x18; Text 'Позиція'
   TextField "Text field_6" at 8,85 size 136x18; Text 'Реперний вимикач'
   TextField "Text field_7" at 8,109 size 80x18; Text 'Швидкість'
   TextField "Text field_8" at 365,133 size 104x18; Text 'Залишок часу'
   IOField "I/O field_1" at 184,54 size 120x32; FormatPattern s999999; Unit  мм
      ProcessValue <- "HMI_DB_Calibration_Trolley_Position_mm"
   IOField "I/O field_2" at 184,102 size 120x32; FormatPattern s9999.99; Unit  об/хв
      ProcessValue <- "HMI_DB_Calibration_Trolley_DriveVelocity_rpm"
   Circle "Circle_49" at 236,86 size 16x16
      Appearance <- "HMI_DB_Calibration_Trolley_Reference3K1"
   TextField "Text field_9" at 47,5 size 240x21; Text 'Статус калібровки мех. візка'
   TextField "Text field_10" at 482,5 size 181x21; Text 'Поточний крок та дія'
   Group "Group_1" at 365,32 size 70x25
   SymbolicIOField "Symbolic I/O field_1" at 453,29 size 327x32; TextOff '0'; TextOn '1'; TextList "TrolleyStepName"
      ProcessValue <- "HMI_DB_Calibration_Trolley_CurrentStep"
   TextField "Text field_11" at 365,85 size 268x18; Text 'Умови переходу на наступний крок:'
   SymbolicIOField "Symbolic I/O field_2" at 365,102 size 416x32; TextOff '0'; TextOn '1'; TextList "TrolleyCondition"
      ProcessValue <- "HMI_DB_Calibration_Trolley_CurrentStep"
   Group "Group_2" at 680,256 size 32x32
   Group "Group_3" at 18,256 size 32x32
   Group "Group_4" at 84,256 size 32x32
   Group "Group_5" at 150,256 size 32x32
   Group "Group_6" at 216,256 size 32x32
   Group "Group_7" at 283,256 size 32x32
   Group "Group_8" at 349,256 size 32x32
   Group "Group_9" at 415,256 size 32x32
   Group "Group_10" at 481,256 size 32x32
   Group "Group_11" at 548,256 size 32x32
   Group "Group_12" at 614,256 size 32x32
   Group "Group_14" at 747,256 size 32x32
   TextField "Text field_23" at 0,295 size 68x28; Text 'Перевірка умов'
   TextField "Text field_25" at 68,295 size 65x40; Text 'Натисніть кнопку "Вперед"'
   TextField "Text field_26" at 133,295 size 67x40; Text 'Рух до реперної точки 3К1'
   TextField "Text field_27" at 198,295 size 69x40; Text 'Відпустіть кнопку "Вперед"'
   TextField "Text field_28" at 263,295 size 85x40; Text 'Перемістить механізм від 3К1'
   TextField "Text field_29" at 330,295 size 70x28; Text 'Відхід завершено'
   TextField "Text field_30" at 399,295 size 65x40; Text 'Натисніть кнопку "Вперед"'
   TextField "Text field_31" at 462,295 size 70x40; Text 'Повторний підхід до 3К1'
   TextField "Text field_32" at 544,295 size 40x28; Text 'Quick Stop'
   TextField "Text field_33" at 593,295 size 75x40; Text 'Очікування зупинки привода'
   TextField "Text field_34" at 665,295 size 62x40; Text 'Запуск preset енкодера'
   TextField "Text field_35" at 725,295 size 75x40; Text 'Калібровку успішно завершено'
   Group "Group_13" at 26,342 size 16x16
   Group "Group_15" at 92,342 size 16x16
   Group "Group_16" at 158,342 size 16x16
   Group "Group_17" at 224,342 size 16x16
   Group "Group_18" at 291,342 size 16x16
   Group "Group_19" at 357,342 size 16x16
   Group "Group_20" at 423,342 size 16x16
   Group "Group_21" at 489,342 size 16x16
   Group "Group_22" at 556,342 size 16x16
   Group "Group_23" at 622,342 size 16x16
   Group "Group_24" at 688,342 size 16x16
   Group "Group_25" at 755,342 size 16x16
   TextField "Text field_36" at 18,381 size 148x18; Text 'Умовні позначення:'
   TextField "Text field_37" at 190,381 size 85x18; Text '- Виконано'
   TextField "Text field_38" at 365,381 size 124x18; Text '- Поточний крок'
   TextField "Text field_39" at 540,381 size 92x18; Text '- Очікується'
   TextField "Text field_40" at 218,226 size 360x21; Text 'Послідовність кроків калібровки мех. візка'
   IOField "I/O field_8" at 540,126 size 60x32; FormatPattern 999; Unit  хв :
      ProcessValue <- "HMI_DB_Calibration_Trolley_TimerRemaining_Min"
   IOField "I/O field_9" at 594,126 size 55x32; FormatPattern 999; Unit  сек
      ProcessValue <- "HMI_DB_Calibration_Trolley_TimerRemaining_Sec"
   Group "Group_26" at 303,58 size 0x25
   TextField "Text field_42" at 8,157 size 88x18; Text 'Інкременти'
   IOField "I/O field_10" at 184,156 size 100x20; FormatPattern s9999999999
      ProcessValue <- "RawPosition"
   Group "Group" at 38,33 size 258x23
   TextField "Text field_43" at 8,133 size 179x18; Text 'Дозвіл від мех. підйому'
   Circle "Circle_53" at 236,134 size 16x16
      Appearance <- "HMI_DB_Calibration_Trolley_PrerequisitesNotOK"
   Circle "Circle_14" at 26,342 size 16x16
      Visibility <- "HMI_DB_Calibration_Trolley_Steps_Active_Step10"
   Circle "Circle_15" at 26,342 size 16x16
      Visibility <- "HMI_DB_Calibration_Trolley_Steps_Completed_Step10"
   Circle "Circle_17" at 92,342 size 16x16
      Visibility <- "HMI_DB_Calibration_Trolley_Steps_Active_Step20"
   Circle "Circle_18" at 92,342 size 16x16
      Visibility <- "HMI_DB_Calibration_Trolley_Steps_Completed_Step20"
   Circle "Circle_20" at 158,342 size 16x16
      Visibility <- "HMI_DB_Calibration_Trolley_Steps_Active_Step30"
   Circle "Circle_21" at 158,342 size 16x16
      Visibility <- "HMI_DB_Calibration_Trolley_Steps_Completed_Step30"
   Circle "Circle_23" at 224,342 size 16x16
      Visibility <- "HMI_DB_Calibration_Trolley_Steps_Active_Step40"
   Circle "Circle_24" at 224,342 size 16x16
      Visibility <- "HMI_DB_Calibration_Trolley_Steps_Completed_Step40"
   Circle "Circle_26" at 291,342 size 16x16
      Visibility <- "HMI_DB_Calibration_Trolley_Steps_Active_Step50"
   Circle "Circle_27" at 291,342 size 16x16
      Visibility <- "HMI_DB_Calibration_Trolley_Steps_Completed_Step50"
   Circle "Circle_29" at 357,342 size 16x16
      Visibility <- "HMI_DB_Calibration_Trolley_Steps_Active_Step60"
   Circle "Circle_30" at 357,342 size 16x16
      Visibility <- "HMI_DB_Calibration_Trolley_Steps_Completed_Step60"
   Circle "Circle_32" at 423,342 size 16x16
      Visibility <- "HMI_DB_Calibration_Trolley_Steps_Active_Step70"
   Circle "Circle_33" at 423,342 size 16x16
      Visibility <- "HMI_DB_Calibration_Trolley_Steps_Completed_Step70"
   Circle "Circle_35" at 489,342 size 16x16
      Visibility <- "HMI_DB_Calibration_Trolley_Steps_Active_Step80"
   Circle "Circle_36" at 489,342 size 16x16
      Visibility <- "HMI_DB_Calibration_Trolley_Steps_Completed_Step80"
   Circle "Circle_38" at 556,342 size 16x16
      Visibility <- "HMI_DB_Calibration_Trolley_Steps_Active_Step90"
   Circle "Circle_39" at 556,342 size 16x16
      Visibility <- "HMI_DB_Calibration_Trolley_Steps_Completed_Step90"
   Circle "Circle_41" at 622,342 size 16x16
      Visibility <- "HMI_DB_Calibration_Trolley_Steps_Active_Step100"
   Circle "Circle_42" at 622,342 size 16x16
      Visibility <- "HMI_DB_Calibration_Trolley_Steps_Completed_Step100"
   Circle "Circle_44" at 688,342 size 16x16
      Visibility <- "HMI_DB_Calibration_Trolley_Steps_Active_Step110"
   Circle "Circle_45" at 688,342 size 16x16
      Visibility <- "HMI_DB_Calibration_Trolley_Steps_Completed_Step110"
   Circle "Circle_47" at 755,342 size 16x16
      Visibility <- "HMI_DB_Calibration_Trolley_Steps_Active_Step130"
   Circle "Circle_48" at 755,342 size 16x16
      Visibility <- "HMI_DB_Calibration_Trolley_Steps_Completed_Step130"
   Line "Line_11" at 303,58 size 0x25
      Visibility <- "HMI_DB_Trolley_movement_mechanism_FirstSpeedForward"
   Line "Line_3" at 303,58 size 0x25
      Visibility <- "HMI_DB_Trolley_movement_mechanism_FirstSpeedBackward"
   TextField "Text field_41" at 83,33 size 169x23; Text 'НЕ КАЛІБРОВАНО'
      Visibility <- "HMI_DB_Calibration_Trolley_Calibrated"
   TextField "Text field_4" at 38,33 size 258x23; Text 'КАЛІБРОВКА АНУЛЬОВАНА'
      Visibility <- "HMI_DB_Calibration_Trolley_Aborted"
   TextField "Text field_2" at 58,33 size 219x23; Text 'КАЛІБРОВКА АКТИВНА'
      Visibility <- "HMI_DB_Calibration_Trolley_Active"
   TextField "Text field_3" at 56,33 size 223x23; Text 'ПОМИЛКА КАЛІБРОВКИ'
      Visibility <- "HMI_DB_Calibration_Trolley_Fault"
   TextField "Text field_1" at 98,33 size 139x23; Text 'КАЛІБРОВАНО'
      Visibility <- "HMI_DB_Calibration_Trolley_Calibrated"

